(* IEC 61131-3 sources: SRCI/RobotLibrary/Library/POUs/General/MC_RobotTask (part 2) *)

END_METHOD

METHOD PRIVATE CreateSendPayload : DINT
VAR_IN_OUT
  /// Robot assignment of function
  AxesGroup                 : AxesGroup;
  /// Outputs of PLC for communication to RC
  RobotOutData              : ARRAY[0..RobotLibraryParameter.ROBOT_OUT_DATA_MAX] OF BYTE;
END_VAR

VAR
  /// internal index
 _idx                       : DINT;
  /// temporary byte
 _tmpByte                   : BYTE;
  /// internal sequence index
 _seqIdx                    : DINT;
  /// internal fragment index
 _fragIdx                   : DINT;
END_VAR

  // ------------------------------------
  // Fill SendData
  // ------------------------------------
  // reset all variables and payload
  SendData.Reset();

  CreateSendPayloadHeader        ( AxesGroup := AxesGroup );
  CreateSendPayloadCyclic        ( AxesGroup := AxesGroup );
  CreateSendPayloadCyclicOptional( AxesGroup := AxesGroup );
  CreateSendPayloadSequence      ( AxesGroup := AxesGroup );
  CreateSendPayloadFooter        ( AxesGroup := AxesGroup );
  CreateSendPayloadLogging       ( AxesGroup := AxesGroup );

  // Copy payload to outputs
  SysDepMemCpy( pDest := ADR(RobotOutData), pSrc := ADR(SendData.Payload), DataLen := RobotLibraryParameter.ROBOT_OUT_DATA_MAX+1);

  // reset NewSEQ flag
  AxesGroup.State.NewSEQ[0] := FALSE; {warning 'Test'}

END_METHOD

METHOD PRIVATE CreateSendPayloadCyclic : DINT
VAR_IN_OUT
  /// Robot assignment of function
  AxesGroup : AxesGroup;
END_VAR

  SendData.AddByte(Telegram.PlcToRob.Cyclic.ToolNo);
  SendData.AddByte(Telegram.PlcToRob.Cyclic.FrameNo);

END_METHOD

METHOD PRIVATE CreateSendPayloadCyclicOptional : DINT
VAR_IN_OUT
  /// Robot assignment of function
  AxesGroup : AxesGroup;
END_VAR

VAR
  /// temporary byte
 _tmpByte   : BYTE;
END_VAR

  // Telegram.PlcToRob.CyclicOptional.SubProgramData {{{
  IF ( AxesGroup.CyclicOptional.PlcToRob.SubProgramData.Active )
  THEN
    SendData.AddDataBlock( ADR(Telegram.PlcToRob.CyclicOptional.SubProgramData.Data), SIZEOF(Telegram.PlcToRob.CyclicOptional.SubProgramData.Data));
  END_IF
  // }}}

  // Telegram.PlcToRob.CyclicOptional.CartesianPos {{{
  IF ( AxesGroup.CyclicOptional.PlcToRob.CartesianPosition.Active)
  THEN
    SendData.AddReal(Telegram.PlcToRob.CyclicOptional.CartesianPosition.X );
    SendData.AddReal(Telegram.PlcToRob.CyclicOptional.CartesianPosition.Y );
    SendData.AddReal(Telegram.PlcToRob.CyclicOptional.CartesianPosition.Z );
    SendData.AddReal(Telegram.PlcToRob.CyclicOptional.CartesianPosition.Rx);
    SendData.AddReal(Telegram.PlcToRob.CyclicOptional.CartesianPosition.Ry);
    SendData.AddReal(Telegram.PlcToRob.CyclicOptional.CartesianPosition.Rz);

   _tmpByte   := 0;
   _tmpByte.0 := Telegram.PlcToRob.CyclicOptional.CartesianPosition.Config.0;
   _tmpByte.1 := Telegram.PlcToRob.CyclicOptional.CartesianPosition.Config.1;
   _tmpByte.2 := Telegram.PlcToRob.CyclicOptional.CartesianPosition.Config.2;

    SendData.AddByte(_tmpByte);

    SendData.AddByte (Telegram.PlcToRob.CyclicOptional.CartesianPosition.Turns_J2_J1             );
    SendData.AddByte (Telegram.PlcToRob.CyclicOptional.CartesianPosition.Turns_J4_J3             );
    SendData.AddByte (Telegram.PlcToRob.CyclicOptional.CartesianPosition.Turns_J6_J5             );
    SendData.AddByte (Telegram.PlcToRob.CyclicOptional.CartesianPosition.Turns_E1                );
    SendData.AddReal (Telegram.PlcToRob.CyclicOptional.CartesianPosition.E1                      );
  END_IF
  // }}}

  // Telegram.PlcToRob.CyclicOptional.JointPosition {{{
  IF ( AxesGroup.CyclicOptional.PlcToRob.JointPosition.Active)
  THEN
    SendData.AddReal(Telegram.PlcToRob.CyclicOptional.JointPosition.J1);
    SendData.AddReal(Telegram.PlcToRob.CyclicOptional.JointPosition.J2);
    SendData.AddReal(Telegram.PlcToRob.CyclicOptional.JointPosition.J3);
    SendData.AddReal(Telegram.PlcToRob.CyclicOptional.JointPosition.J4);
    SendData.AddReal(Telegram.PlcToRob.CyclicOptional.JointPosition.J5);
    SendData.AddReal(Telegram.PlcToRob.CyclicOptional.JointPosition.J6);
    SendData.AddReal(Telegram.PlcToRob.CyclicOptional.JointPosition.E1);
  END_IF
  // }}}

  // Telegram.PlcToRob.CyclicOptional.Force {{{
  IF ( AxesGroup.CyclicOptional.PlcToRob.Force.Active)
  THEN
    SendData.AddReal(Telegram.PlcToRob.CyclicOptional.Force.X);
    SendData.AddReal(Telegram.PlcToRob.CyclicOptional.Force.Y);
    SendData.AddReal(Telegram.PlcToRob.CyclicOptional.Force.Z);
    SendData.AddReal(Telegram.PlcToRob.CyclicOptional.Force.Rx);
    SendData.AddReal(Telegram.PlcToRob.CyclicOptional.Force.Ry);
    SendData.AddReal(Telegram.PlcToRob.CyclicOptional.Force.Rz);
  END_IF
  // }}}

  // Telegram.PlcToRob.CyclicOptional.TwoSequences {{{
  // }}}

  // AxesGroup.OptionalCyclic.PlcToRob.CartesianPosExt {{{
  IF ( AxesGroup.CyclicOptional.PlcToRob.CartesianPositionExt.Active)
  THEN
    SendData.AddReal(Telegram.PlcToRob.CyclicOptional.CartesianPositionExt.E2);
    SendData.AddReal(Telegram.PlcToRob.CyclicOptional.CartesianPositionExt.E3);
    SendData.AddReal(Telegram.PlcToRob.CyclicOptional.CartesianPositionExt.E4);
    SendData.AddReal(Telegram.PlcToRob.CyclicOptional.CartesianPositionExt.E5);
    SendData.AddReal(Telegram.PlcToRob.CyclicOptional.CartesianPositionExt.E6);
  END_IF
  // }}}

  // AxesGroup.OptionalCyclic.PlcToRob.JointPositionExt {{{
  IF ( AxesGroup.CyclicOptional.PlcToRob.JointPositionExt.Active)
  THEN
    SendData.AddReal(Telegram.PlcToRob.CyclicOptional.JointPositionExt.E2);
    SendData.AddReal(Telegram.PlcToRob.CyclicOptional.JointPositionExt.E3);
    SendData.AddReal(Telegram.PlcToRob.CyclicOptional.JointPositionExt.E4);
    SendData.AddReal(Telegram.PlcToRob.CyclicOptional.JointPositionExt.E5);
    SendData.AddReal(Telegram.PlcToRob.CyclicOptional.JointPositionExt.E6);
  END_IF
  // }}}

  // Telegram.PlcToRob.CyclicOptional..CartesianForceExt {{{
  IF ( AxesGroup.CyclicOptional.PlcToRob.ForceExt.Active)
  THEN
    SendData.AddReal(Telegram.PlcToRob.CyclicOptional.ForceExt.E1);
    SendData.AddReal(Telegram.PlcToRob.CyclicOptional.ForceExt.E2);
    SendData.AddReal(Telegram.PlcToRob.CyclicOptional.ForceExt.E3);
    SendData.AddReal(Telegram.PlcToRob.CyclicOptional.ForceExt.E4);
    SendData.AddReal(Telegram.PlcToRob.CyclicOptional.ForceExt.E5);
    SendData.AddReal(Telegram.PlcToRob.CyclicOptional.ForceExt.E6);
  END_IF
  // }}}

END_METHOD

METHOD PRIVATE CreateSendPayloadFooter : DINT
VAR_IN_OUT
  /// Robot assignment of function
  AxesGroup : AxesGroup;
END_VAR
VAR
  /// index of lifesign in footer
  _lifeSignIdxFooter : DINT;
END_VAR

  IF (( _parCfg.Com.TelegramLengthPlcToRob    >= 1                                           ) AND
      ( _parCfg.Com.TelegramLengthPlcToRob    <= RobotLibraryParameter.ROBOT_OUT_DATA_MAX +1 ))
  THEN
    // set index of life sign byte
   _lifeSignIdxFooter := _parCfg.Com.TelegramLengthPlcToRob -1;

    SendData.Payload[_lifeSignIdxFooter] := AxesGroup.Cyclic.PlcToRob.LifeSign;
  END_IF

END_METHOD

METHOD PRIVATE CreateSendPayloadHeader : DINT
VAR_IN_OUT
  /// Robot assignment of function
  AxesGroup : AxesGroup;
END_VAR

  SendData.AddByte(Telegram.PlcToRob.Header.SRCIVersion           );
  SendData.AddByte(Telegram.PlcToRob.Header.FastStop_LifeSign     );
  SendData.AddUint(Telegram.PlcToRob.Header.TelegramLengthPlcToRob);
  SendData.AddUint(Telegram.PlcToRob.Header.TelegramLengthRobToPlc);
  SendData.AddByte(Telegram.PlcToRob.Header.AxesGroupID_Control   );
  SendData.AddByte(Telegram.PlcToRob.Header.Reserved              );
  SendData.AddUint(Telegram.PlcToRob.Header.TelegramNumberPlcToRob);
  SendData.AddUint(Telegram.PlcToRob.Header.TelegramNumberRobToPlc);
  SendData.AddUint(Telegram.PlcToRob.Header.ClientDate            );
  SendData.AddTime(Telegram.PlcToRob.Header.ClientTime            );

END_METHOD

METHOD PRIVATE CreateSendPayloadLogging : DINT
VAR_IN_OUT
  /// Robot assignment of function
  AxesGroup                 : AxesGroup;
END_VAR

  IF  ((( Telegram.PlcToRob.Sequence[0].Header.PayloadLength > 0 ) AND (AxesGroup.State.NewSEQ[0] )) OR
       (( Telegram.PlcToRob.Sequence[1].Header.PayloadLength > 0 ) AND (AxesGroup.State.NewSEQ[1] )))
  THEN
    // Create log entry
    CreateLogMessagePara1 ( Timestamp   := SystemTime,
                            MessageType := MessageType.CMD,
                            Severity    := Severity.DEBUG,
                            MessageCode := 0,
                            MessageText := 'SendData: Bytes send in total: {1}',
                            Para1       :=  UDINT_TO_STRING(SendData.PayloadLen));
  END_IF

END_METHOD

METHOD PRIVATE CreateSendPayloadSequence : DINT
VAR_IN_OUT
  /// Robot assignment of function
  AxesGroup                 : AxesGroup;
END_VAR

VAR
  /// internal sequence index
 _seqIdx                    : DINT;
  /// internal fragment index
 _fragIdx                   : DINT;
END_VAR

  FOR _seqIdx := 0 TO AxesGroup.State.SequenceCountSend
  DO
    // Check 2nd sequence ? -> goto 2nd sequence payload address
    IF ( _seqIdx = SECONDARY_SEQUENCE )
    THEN
      SendData.PayloadPtr := CalculateSequencePayloadStartAdr(AxesGroup := AxesGroup,
                                                              Direction := ComDirection.PLC_TO_ROB,
                                                              Sequence  := SequenceFlag.SECONDARY_SEQUENCE);
    END_IF

    // Telegram.PlcToRob.Sequence[x].Header {{{
    SendData.AddUint(Telegram.PlcToRob.Sequence[_seqIdx].Header.SEQ_ACK);
    SendData.AddUint(Telegram.PlcToRob.Sequence[_seqIdx].Header.PayloadLength);
    // }}}

    // check limit reachted ?
    IF ( SendData.PayloadPtr + FOOTER_SIZE >= Telegram.PlcToRob.Header.TelegramLengthPlcToRob)
    THEN
      EXIT;
    END_IF

    // PlcToRob.Sequence[x].Fragment[x] {{{
    FOR _fragIdx := 0 TO AxesGroup.State.FragmentCountSend[_seqIdx]
    DO

      IF (Telegram.PlcToRob.Sequence[_seqIdx].Fragment[_fragIdx].Header.PayloadLength > 0)
      THEN
        // PlcToRob.Sequence[x].Fragment[x].Header {{{
        SendData.AddUint(Telegram.PlcToRob.Sequence[_seqIdx].Fragment[_fragIdx].Header.CmdID);
        SendData.AddByte(Telegram.PlcToRob.Sequence[_seqIdx].Fragment[_fragIdx].Header.Reserve);
        SendData.AddByte(Telegram.PlcToRob.Sequence[_seqIdx].Fragment[_fragIdx].Header.FragmentAction);
        SendData.AddUint(Telegram.PlcToRob.Sequence[_seqIdx].Fragment[_fragIdx].Header.PayloadPointer);
        SendData.AddUint(Telegram.PlcToRob.Sequence[_seqIdx].Fragment[_fragIdx].Header.PayloadLength);
        // }}}

        // PlcToRob.Sequence[x].Fragment[x].Command {{{

        // Hint: the command header is part of the fragment payload
        IF (Telegram.PlcToRob.Sequence[_seqIdx].Fragment[_fragIdx].Header.PayloadLength > 0)
        THEN
          SendData.AddDataBlock( pValue :=  ADR(Telegram.PlcToRob.Sequence[_seqIdx].Fragment[_fragIdx].Command.Payload           ) + Telegram.PlcToRob.Sequence[_seqIdx].Fragment[_fragIdx].Header.PayloadPointer,
                                   Size :=     (Telegram.PlcToRob.Sequence[_seqIdx].Fragment[_fragIdx].Header.PayloadLength      ));

        END_IF

        IF (SendData.PayloadLen = 232)
        THEN
          SendData.PayloadLen := SendData.PayloadLen;
  			END_IF

      END_IF
      // }}}
    END_FOR
    // }}}
  END_FOR

END_METHOD

METHOD FB_init : BOOL
VAR_INPUT
  bInitRetains : BOOL; // if TRUE, the retain variables are initialized (warm start / cold start)
  bInCopyCode : BOOL;  // if TRUE, the instance afterwards gets moved into the copy code (online change)
END_VAR

  MyType := 'MC_RobotTaskFB';

  // Create log entry
  CreateLogMessage ( Timestamp   := SystemTime,
                     MessageType := MessageType.CMD,
                     Severity    := Severity.DEBUG,
                     MessageCode := 0,
                     MessageText := 'PLC started / restarted');

END_METHOD

METHOD PRIVATE HandleAliveBit
VAR_INPUT
  LifeSign : BYTE;
END_VAR

VAR_INST
  /// flag that indicates that the 1st cyclce is running
  First : BOOL := TRUE;
END_VAR

  IF (First AND LifeSign > 0)
  THEN
    // init alive value
   _aliveValue := LifeSign;
    // reset first flag
    First := FALSE;
  END_IF

  _aliveCheck ( IN  := (_aliveValue = LifeSign) , PT := ParCfg.Com.LifeSignTimeOut + ParCfg.Plc.CycleTime);
  _alive_R    ( CLK := _aliveBit);
  _alive_F    ( CLK := _aliveBit);

  IF ( _aliveValue <> LifeSign)
  THEN
   _aliveValue := LifeSign;
   _aliveBit   := TRUE;
  END_IF

  IF (_aliveCheck.Q)
  THEN
   _aliveBit := FALSE;
  END_IF

  IF (_alive_R.Q)
  THEN
    // Create log entry
    CreateLogMessage ( Timestamp   := SystemTime,
                       MessageType := MessageType.CMD,
                       Severity    := Severity.INFO,
                       MessageCode := 0,
                       MessageText := 'Data Exchange is running (Alive-Bit)');
  END_IF

  IF (_alive_F.Q)
  THEN
    // Create log entry
    CreateLogMessage ( Timestamp   := SystemTime,
                       MessageType := MessageType.CMD,
                       Severity    := Severity.INFO,
                       MessageCode := 0,
                       MessageText := 'Data Exchange has stopped (Alive-Bit)');
  END_IF

END_METHOD

METHOD PRIVATE HandleAxesGroup
VAR_IN_OUT
  /// Robot assignment of function
  AxesGroup : AxesGroup;
END_VAR

  HandleAxesGroupAcyclic       ( AxesGroup    := AxesGroup);
  HandleAxesGroupCyclic        ( AxesGroup    := AxesGroup);
  HandleAxesGroupCyclicOptional( AxesGroup    := AxesGroup);
  HandleAxesGroupMessageLog    ( AxesGroup    := AxesGroup);
  HandleAxesGroupParameter     ( AxesGroup    := AxesGroup);
  HandleAxesGroupState         ( AxesGroup    := AxesGroup);

END_METHOD

METHOD PRIVATE HandleAxesGroupAcyclic
VAR_IN_OUT
  /// Robot assignment of function
  AxesGroup : AxesGroup;
END_VAR

  // Call active command register FB
  AxesGroup.Acyclic.ActiveCommandRegister(SystemTime     := SystemTime,
                                          RegisterSize   := MIN( RobotLibraryParameter.ACTIVE_CMD_REGISTER_ENTRIES_MAX, AxesGroup.Parameter.Rob.Parameter.LengthACR),
                                          InternalLogger := AxesGroup.MessageLog,
                                          ExternalLogger := AxesGroup.MessageLog.ExternalLogger,
                                          LogLevel       := AxesGroup.MessageLog.LogLevel);

END_METHOD

METHOD PRIVATE HandleAxesGroupCyclic
VAR_IN_OUT
  /// Robot assignment of function
  AxesGroup : AxesGroup;
END_VAR

  // set instance AxesGroupID
  AxesGroup.Cyclic.PlcToRob.AxesGroupID := AxesGroupID;
  // Set Version
  AxesGroup.Cyclic.PlcToRob.SRCIVersion := RobotLibraryConstants.SRCIVersion;

  AxesGroup.Cyclic.PlcToRob.TelegramLengthPlcToRob := _parCfg.Com.TelegramLengthPlcToRob;
  AxesGroup.Cyclic.PlcToRob.TelegramLengthRobToPlc := _parCfg.Com.TelegramLengthRobToPlc;

  AxesGroup.Cyclic.PlcToRob.TelegramNumberPlcToRob := PlcOptionalCyclicToUint(AxesGroup.Parameter.Plc.OptionalCyclic);
  AxesGroup.Cyclic.PlcToRob.TelegramNumberRobToPlc := RobOptionalCyclicToUint(AxesGroup.Parameter.Rob.OptionalCyclic);

  // Set Date + Time
  AxesGroup.Cyclic.PlcToRob.ClientDate  := DATE_TO_IEC_DATE(SystemTime.SystemDate);
  AxesGroup.Cyclic.PlcToRob.ClientTime  := TIME_TO_IEC_TIME(SystemTime.SystemTime);

END_METHOD

METHOD PRIVATE HandleAxesGroupCyclicOptional
VAR_IN_OUT
  /// Robot assignment of function
  AxesGroup : AxesGroup;
END_VAR

  // PlcToRob {{{
  AxesGroup.CyclicOptional.PlcToRob.SubProgramData      .Active := AxesGroup.Parameter.Plc.OptionalCyclic.UseCallSubprogram;
  AxesGroup.CyclicOptional.PlcToRob.CartesianPosition   .Active := AxesGroup.Parameter.Plc.OptionalCyclic.UseCartesianPosition;
  AxesGroup.CyclicOptional.PlcToRob.JointPosition       .Active := AxesGroup.Parameter.Plc.OptionalCyclic.UseJointPosition;
  AxesGroup.CyclicOptional.PlcToRob.Force               .Active := AxesGroup.Parameter.Plc.OptionalCyclic.UseForce;
  AxesGroup.CyclicOptional.PlcToRob.CartesianPositionExt.Active := AxesGroup.Parameter.Plc.OptionalCyclic.UseCartesianPositionExt;
  AxesGroup.CyclicOptional.PlcToRob.JointPositionExt    .Active := AxesGroup.Parameter.Plc.OptionalCyclic.UseJointPositionExt;
  // }}}

  // RobToPlc {{{
  AxesGroup.CyclicOptional.RobToPlc.SubProgramData      .Active := AxesGroup.Parameter.Rob.OptionalCyclic.UseCallSubprogram;
  AxesGroup.CyclicOptional.RobToPlc.CartesianPosition   .Active := AxesGroup.Parameter.Rob.OptionalCyclic.UseCartesianPosition;
  AxesGroup.CyclicOptional.RobToPlc.JointPosition       .Active := AxesGroup.Parameter.Rob.OptionalCyclic.UseJointPosition;
  AxesGroup.CyclicOptional.RobToPlc.Force               .Active := AxesGroup.Parameter.Rob.OptionalCyclic.UseForce;
  AxesGroup.CyclicOptional.RobToPlc.Current             .Active := AxesGroup.Parameter.Rob.OptionalCyclic.UseCurrent;
  AxesGroup.CyclicOptional.RobToPlc.CartesianPositionExt.Active := AxesGroup.Parameter.Rob.OptionalCyclic.UseCartesianPositionExt;
  AxesGroup.CyclicOptional.RobToPlc.JointPositionExt    .Active := AxesGroup.Parameter.Rob.OptionalCyclic.UseJointPositionExt;
  AxesGroup.CyclicOptional.RobToPlc.ForceExt            .Active := AxesGroup.Parameter.Rob.OptionalCyclic.UseForceExt;
  AxesGroup.CyclicOptional.RobToPlc.CurrentExt          .Active := AxesGroup.Parameter.Rob.OptionalCyclic.UseCurrentExt;
  // }}}

END_METHOD

METHOD PRIVATE HandleAxesGroupMessageLog
VAR_IN_OUT
  /// Robot assignment of function
  AxesGroup  : AxesGroup;
END_VAR

  // Set External logger
  AxesGroup.MessageLog.ExternalLogger := ExternalLogger;
  AxesGroup.MessageLog.LogLevel       := LogLevel;

  IF (AxesGroup.State.GroupReset_R.Q)
  THEN
    AxesGroup.MessageLog.DeleteMessages();
    AxesGroup.MessageLog.DeleteSystemLogs();
  END_IF

END_METHOD

METHOD PRIVATE HandleAxesGroupParameter
VAR_IN_OUT
  /// Robot assignment of function
  AxesGroup : AxesGroup;
END_VAR

  IF (_exchangeConfiguration.Enabled)
  THEN
    AxesGroup.Parameter.Plc.Parameter                           := _parCfg.Plc.Parameter;
    AxesGroup.Parameter.Plc.OptionalCyclic                      := _parCfg.Plc.OptionalCyclic;
    AxesGroup.Parameter.Rob.OptionalCyclic                      := _parCfg.Rob.OptionalCyclic;

    AxesGroup.Parameter.Rob.Parameter.LengthACR                 := _exchangeConfiguration.OutCmd.LengthACR;
    AxesGroup.Parameter.Rob.Parameter.HighestToolIndex          := _exchangeConfiguration.OutCmd.HighestToolIndex;
    AxesGroup.Parameter.Rob.Parameter.HighestFrameIndex         := _exchangeConfiguration.OutCmd.HighestFrameIndex;
    AxesGroup.Parameter.Rob.Parameter.HighestLoadIndex          := _exchangeConfiguration.OutCmd.HighestLoadIndex;
    AxesGroup.Parameter.Rob.Parameter.HighestWorkAreaIndex      := _exchangeConfiguration.OutCmd.HighestWorkAreaIndex;
    AxesGroup.Parameter.Rob.Parameter.DataInSync                := _exchangeConfiguration.OutCmd.DataInSync;
    AxesGroup.Parameter.Rob.Parameter.ChangeIndexTool           := _exchangeConfiguration.OutCmd.ChangeIndexTool;
    AxesGroup.Parameter.Rob.Parameter.ChangeIndexFrame          := _exchangeConfiguration.OutCmd.ChangeIndexFrame;
    AxesGroup.Parameter.Rob.Parameter.ChangeIndexLoad           := _exchangeConfiguration.OutCmd.ChangeIndexLoad;
    AxesGroup.Parameter.Rob.Parameter.ChangeIndexWorkArea       := _exchangeConfiguration.OutCmd.ChangeIndexWorkArea;
    AxesGroup.Parameter.Rob.Parameter.RAWorkingHours            := _exchangeConfiguration.OutCmd.RAWorkingHours;
    AxesGroup.Parameter.Rob.Parameter.BrakeTestRequired         := _exchangeConfiguration.OutCmd.BrakeTestRequired;
    AxesGroup.Parameter.Rob.Parameter.StepModeExactStopActive   := _exchangeConfiguration.OutCmd.StepModeExactStopActive;
    AxesGroup.Parameter.Rob.Parameter.StepModeBlendingActive    := _exchangeConfiguration.OutCmd.StepModeBlendingActive;
    AxesGroup.Parameter.Rob.Parameter.PathAccuracyMode          := _exchangeConfiguration.OutCmd.PathAccuracyMode;
    AxesGroup.Parameter.Rob.Parameter.AvoidSingularity          := _exchangeConfiguration.OutCmd.AvoidSingularity;
    AxesGroup.Parameter.Rob.Parameter.CollisionDetectionEnabled := _exchangeConfiguration.OutCmd.CollisionDetectionEnabled;
    AxesGroup.Parameter.Rob.Parameter.AcceleratingSupported     := _exchangeConfiguration.OutCmd.AcceleratingSupported;
    AxesGroup.Parameter.Rob.Parameter.DecceleratingSupported    := _exchangeConfiguration.OutCmd.DecceleratingSupported;
    AxesGroup.Parameter.Rob.Parameter.ConstantVelocitySupported := _exchangeConfiguration.OutCmd.ConstantVelocitySupported;
    AxesGroup.Parameter.Rob.Parameter.RCWorkingHours            := _exchangeConfiguration.OutCmd.RCWorkingHours;
  ELSE
    AxesGroup.Parameter.Plc.Parameter                           := ParCfg.Plc.Parameter;
    AxesGroup.Parameter.Plc.OptionalCyclic                      := ParCfg.Plc.OptionalCyclic;
    AxesGroup.Parameter.Rob.OptionalCyclic                      := ParCfg.Rob.OptionalCyclic;
  END_IF

END_METHOD

METHOD PRIVATE HandleAxesGroupState
VAR_IN_OUT
  /// Robot assignment of function
  AxesGroup : AxesGroup;
END_VAR
VAR
  /// internal index for loops
 _idx       : DINT;
END_VAR

  AxesGroup.State.AliveOk      := _aliveBit;
  AxesGroup.State.Initialized  := Initialized  AND AxesGroup.State.AliveOk;
  AxesGroup.State.Synchronized := Synchronized AND AxesGroup.State.AliveOk;
  AxesGroup.State.CMDsEnabled  := AxesGroup.State.Initialized OR
                                  AxesGroup.State.Synchronized;

  AxesGroup.State.ConfigExchanged := _exchangeConfiguration.Enabled;

  AxesGroup.State.UnifiedFrameIndex                    := DINT_TO_USINT( MIN( RobotLibraryParameter.FRAME_MAX -1    , _exchangeConfiguration.OutCmd.HighestFrameIndex   ));
  AxesGroup.State.UnifiedToolIndex                     := DINT_TO_USINT( MIN( RobotLibraryParameter.TOOL_MAX -1     , _exchangeConfiguration.OutCmd.HighestToolIndex    ));
  AxesGroup.State.UnifiedLoadIndex                     := DINT_TO_USINT( MIN( RobotLibraryParameter.LOAD_MAX-1      , _exchangeConfiguration.OutCmd.HighestLoadIndex    ));
  AxesGroup.State.UnifiedWorkAreaIndex                 := DINT_TO_USINT( MIN( RobotLibraryParameter.WORK_AREAS_MAX-1, _exchangeConfiguration.OutCmd.HighestWorkAreaIndex));

  AxesGroup.State.DataEnableSync                       := _exchangeConfiguration.ParCmd.DataEnableSync;
  AxesGroup.State.SyncStateRc.InSync.Frame             := _exchangeConfiguration.OutCmd.DataInSync.FramesInSync;
  AxesGroup.State.SyncStateRc.InSync.Tool              := _exchangeConfiguration.OutCmd.DataInSync.ToolsInSync;
  AxesGroup.State.SyncStateRc.InSync.Load              := _exchangeConfiguration.OutCmd.DataInSync.LoadsInSync;
  AxesGroup.State.SyncStateRc.InSync.WorkArea          := _exchangeConfiguration.OutCmd.DataInSync.WorkAreasInSync;
  AxesGroup.State.SyncStateRc.InSync.SwLimits          := _exchangeConfiguration.OutCmd.DataInSync.SoftwareLimitsInSync;
  AxesGroup.State.SyncStateRc.InSync.DefaultDynamics   := _exchangeConfiguration.OutCmd.DataInSync.DefaultDynamicsInSync;
  AxesGroup.State.SyncStateRc.InSync.ReferenceDynamics := _exchangeConfiguration.OutCmd.DataInSync.ReferenceDynamicsInSync;

  AxesGroup.State.SyncStateRc.UnSyncNo.Frame           := _exchangeConfiguration.OutCmd.ChangeIndexFrame;
  AxesGroup.State.SyncStateRc.UnSyncNo.Tool            := _exchangeConfiguration.OutCmd.ChangeIndexTool;
  AxesGroup.State.SyncStateRc.UnSyncNo.Load            := _exchangeConfiguration.OutCmd.ChangeIndexLoad;
  AxesGroup.State.SyncStateRc.UnSyncNo.WorkArea        := _exchangeConfiguration.OutCmd.ChangeIndexWorkArea;

  // Update internal data
  AxesGroup.State.SystemTime   := SystemTime;
  AxesGroup.State.OnlineChange := OnlineChange;
  AxesGroup.State.Initialized  := Initialized;

  // Create rising and falling edges for Online Change
  AxesGroup.State.OnlineChange_R(CLK := OnlineChange);
  AxesGroup.State.OnlineChange_F(CLK := OnlineChange);

  // Create rising and falling edges for GroupReset
  AxesGroup.State.GroupReset_R(CLK := AxesGroup.State.GroupReset);
  AxesGroup.State.GroupReset_F(CLK := AxesGroup.State.GroupReset);

  // Copy function block results
  AxesGroup.State.RobotData         := _readRobotData.OutCmd;
  AxesGroup.State.ConfigurationData := _exchangeConfiguration.OutCmd;

END_METHOD

METHOD PRIVATE HandleInvalidFrames
VAR_IN_OUT
   /// Robot assignment of function
  AxesGroup   : AxesGroup;
    /// Inputs of PLC for communication from RC
  RobotInData : ARRAY[0..RobotLibraryParameter.ROBOT_IN_DATA_MAX ] OF BYTE;
END_VAR
VAR
  /// index of lifesign in header
 _lifeSignIdxHeader : DINT;
  /// Value of lifesign in header
 _lifeSignHeader    : BYTE;
  /// index of lifesign in footer
 _lifeSignIdxFooter : DINT;
  /// Value of lifesign in footer
 _lifeSignFooter    : BYTE;
END_VAR
VAR_INST
  /// Timeout for invalid frames counter check
 _invalidFrameCounterCheck_D : TON;
  /// last count of invalid frames
 _lastInvalidFrames          : UDINT;
END_VAR

  IF (( _parCfg.Com.TelegramLengthRobToPlc     < 1                                       ) AND
      ( _parCfg.Com.TelegramLengthRobToPlc - 1 > RobotLibraryParameter.ROBOT_IN_DATA_MAX ))
  THEN
    // no valid telegram length settings
    RETURN;
  END_IF

  // set index of last byte
  _lifeSignIdxHeader := 1;
  _lifeSignIdxFooter := _parCfg.Com.TelegramLengthRobToPlc -1;

  IF ( AxesGroup.Cyclic.RobToPlc.TelegramState = TelegramState.INITIALIZED )
  THEN
    // Get lifesign values
   _lifeSignHeader := GetHalfeByteHi( RobotInData[_lifeSignIdxHeader]);
   _lifeSignFooter := GetHalfeByteHi( RobotInData[_lifeSignIdxFooter]);
  END_IF

  // Timer for invalid frame(s) message
  _invalidFrameCounterCheck_D( IN := TRUE , PT := RobotLibraryParameter.INVALID_FRAMES_CHECK_TIMEOUT);

  // Check Frame is valid :
  // ----------------------
  IF ( _lifeSignHeader <> _lifeSignFooter )
  THEN
    AxesGroup.State.InvalidFrames := AxesGroup.State.InvalidFrames + 1;
  END_IF

  // Check timeout for invalid frame message
  IF ( _invalidFrameCounterCheck_D.Q )
  THEN
    // reset timer
   _invalidFrameCounterCheck_D( IN := FALSE);

    // compare invalid frame(s) counter
    IF ( AxesGroup.State.InvalidFrames <> _lastInvalidFrames)
    THEN
      // store last invalid frame(s) counter value
     _lastInvalidFrames := AxesGroup.State.InvalidFrames;
      // Create log entry
      CreateLogMessagePara1 ( Timestamp   := SystemTime,
                              MessageType := MessageType.CMD,
                              Severity    := Severity.WARNING,
                              MessageCode := 0,
                              MessageText := 'Detected invalid frames {1} in total',
                              Para1       :=  UDINT_TO_STRING(AxesGroup.State.InvalidFrames));
    END_IF
  END_IF

  // Reset invalid frames counter with rising edge of group reset
  IF ( AxesGroup.State.GroupReset_R.Q)
  THEN
    AxesGroup.State.InvalidFrames := 0;
               _lastInvalidFrames := 0;

    // Create log entry
    CreateLogMessage ( Timestamp   := SystemTime,
                       MessageType := MessageType.CMD,
                       Severity    := Severity.INFO,
                       MessageCode := 0,
                       MessageText := 'Reset invalid frames counter by executing GroupReset');
  END_IF

END_METHOD

METHOD PRIVATE HandleLifeSign
VAR_IN_OUT
  /// Robot assignment of function
  AxesGroup    : AxesGroup;
END_VAR
VAR_INST
  /// flag for 1st cycle
 _first : BOOL := TRUE;
END_VAR

  IF ( _first ) OR ( NOT Enable )
  THEN
    // init LifeSign
    AxesGroup.Cyclic.PlcToRob.LifeSign := 0;
    // reset first flag
   _first := FALSE;
    // prevent inc LifeSign in the 1st cycle (Code below)
    RETURN;
  END_IF

  AxesGroup.Cyclic.PlcToRob.LifeSign := AxesGroup.Cyclic.PlcToRob.LifeSign + 1;

  IF ( AxesGroup.Cyclic.PlcToRob.LifeSign > 15 )
  THEN
    AxesGroup.Cyclic.PlcToRob.LifeSign := 1; // 0 is only in the very 1st cycle to indicate the system start in logging
  END_IF

  IF ( Enable ) AND ( _alive_F.Q )
  THEN
    // Reset initialized flag
    Initialized := FALSE;
    // Reset Synchronized flag
    Synchronized := FALSE;

    // Set error
    ErrorID := RobotLibraryErrorIdEnum.ERR_CONNECTION_LOST;
    // Create log entry
    CreateLogMessage ( Timestamp   := SystemTime,
                       MessageType := MessageType.CMD,
                       Severity    := Severity.FATAL_ERROR,
                       MessageCode := 0,
                       MessageText := 'LifeSign timeout -> Reinitialization required !');
  END_IF

  // Reset connection lost error
  IF ( NOT Enable ) AND ( _aliveBit ) AND ( ErrorID = RobotLibraryErrorIdEnum.ERR_CONNECTION_LOST )
  THEN
    ErrorID := 0;
  END_IF

END_METHOD

METHOD HandleLogMessagesAck
VAR_IN_OUT
   /// Robot assignment of function
  AxesGroup : AxesGroup;
END_VAR

  IF (( _readMessages.Enabled           ) AND
      ( _readMessages.OutCmd.MsgId > 0  ))
  THEN
    // Check if message has been entered into the message log ?
    IF ( AxesGroup.MessageLog.CheckMessageCodePresent(_readMessages.OutCmd.ErrorCode ))
    THEN
      // Set Message ID as Acknowlege ID
     _readMessages.ParCmd.MsgID := _readMessages.OutCmd.MsgId;
  	END_IF
  END_IF

END_METHOD

METHOD PRIVATE HandleSeqAck
VAR_IN_OUT
   /// Robot assignment of function
  AxesGroup    : AxesGroup;
END_VAR
VAR
  /// internal index for loops
 _idx : DINT;
END_VAR

  FOR _idx := 0 TO  AxesGroup.State.SequenceCountSend
  DO
    AxesGroup.State.CurrentAck[_idx] := Telegram.RobToPlc.Sequence[_idx].Header.SEQ_ACK;

    IF (NOT Enable)
    THEN
      AxesGroup.State.CurrentSEQ[0] := 0;
      AxesGroup.State.CurrentSEQ[1] := 0;
    END_IF

    // Check Seq/Ack :
    // ----------------------
    IF ( AxesGroup.State.CurrentAck[_idx] = AxesGroup.State.CurrentSEQ[_idx] )
    THEN
      AxesGroup.State.CurrentSEQ[_idx] := MAX(AxesGroup.State.CurrentSEQ[0],AxesGroup.State.CurrentSEQ[1]) +1;

      IF (AxesGroup.State.CurrentSEQ[_idx] >= 255) {warning 'ToDo: Test for Yaskawa'}
      THEN
        AxesGroup.State.CurrentSEQ[_idx] := 0;
  		END_IF

      AxesGroup.State.NewSEQ[_idx] := TRUE;
    END_IF
  END_FOR

END_METHOD

METHOD PRIVATE HandleSync
VAR_IN_OUT
   /// Robot assignment of function
  AxesGroup : AxesGroup;
  /// ToolData stored on PLC.For more information refer to 5.5.6.4
  ToolData          : ARRAY[0..RobotLibraryParameter.TOOL_MAX -1      ] OF Tool;
  /// LoadData stored on PLC.For more information refer to 5.5.6.4
  FrameData         : ARRAY[0..RobotLibraryParameter.FRAME_MAX -1     ] OF Frame;
  /// LoadData stored on PLC.For more information refer to 5.5.6.4
  LoadData          : ARRAY[0..RobotLibraryParameter.LOAD_MAX -1      ] OF Load;
  /// Work areas stored on PLC. For more information refer to 5.5.8
  WorkAreas         : ARRAY[0..RobotLibraryParameter.WORK_AREAS_MAX -1] OF RobotWorkArea;
  /// Software limits stored on PLC
  SWLimits          : SWLimits;
  /// Default dynamics stored on PLC. For more information refer to 5.5.7
  DefaultDynamics   : DefaultDynamics;
  /// Reference dynamics stored on PLC. For more information refer to 5.5.7
  ReferenceDynamics : ReferenceDynamics;
END_VAR

VAR
  /// flag that indicates at least any iten has enabled synchronisation
 _dataEnableSyncAny        : BOOL;
  /// flag that indicates that the frame datas are synchronized or deactivated
 _inSyncFrameOk            : BOOL;
  /// flag that indicates that the tool datas are synchronized or deactivated
 _inSyncToolOk             : BOOL;
  /// flag that indicates that the load datas are synchronized or deactivated
 _inSyncLoadOk             : BOOL;
  /// flag that indicates that the work areas are synchronized or deactivated
 _inSyncWorkAreaOk         : BOOL;
  /// flag that indicates that the SW limits are synchronized or deactivated
 _inSyncSwLimitsOk         : BOOL;
  /// flag that indicates that the default dynamice are synchronized or deactivated
 _inSyncDefaultDynamicOk   : BOOL;
  /// flag that indicates that the reference dynamice are synchronized or deactivated
 _InSyncReferenceDynamicOk : BOOL;
END_VAR

  HandleSyncToolData              ( AxesGroup := AxesGroup, ToolData          := ToolData);
  //RETURN; {warning 'ToDo: Enable Sync again'}

  HandleSyncFrameData             ( AxesGroup := AxesGroup, FrameData         := FrameData);
  HandleSyncLoadData              ( AxesGroup := AxesGroup, LoadData          := LoadData);
  HandleSyncRobotDefaultDynamics  ( AxesGroup := AxesGroup, DefaultDynamics   := DefaultDynamics);
  HandleSyncRobotReferenceDynamics( AxesGroup := AxesGroup, ReferenceDynamics := ReferenceDynamics);
  HandleSyncRobotSWLimits         ( AxesGroup := AxesGroup, SwLimits          := SwLimits);
  HandleSyncToolData              ( AxesGroup := AxesGroup, ToolData          := ToolData);
  HandleSyncWorkArea              ( AxesGroup := AxesGroup, WorkAreas         := WorkAreas);

  // check any synchronisation activated ?
  _dataEnableSyncAny :=        ((     AxesGroup.State.DataEnableSync.EnableSyncFrame             )  OR
                                (     AxesGroup.State.DataEnableSync.EnableSyncTool              )  OR
                                (     AxesGroup.State.DataEnableSync.EnableSyncLoad              )  OR
                                (     AxesGroup.State.DataEnableSync.EnableSyncWorkArea          )  OR
                                (     AxesGroup.State.DataEnableSync.EnableSyncSWLimits          )  OR
                                (     AxesGroup.State.DataEnableSync.EnableSyncDefaultDynamics   )  OR
                                (     AxesGroup.State.DataEnableSync.EnableSyncReferenceDynamics ));

  _inSyncFrameOk :=            ((     AxesGroup.State.SyncStatePlc     .InSync.Frame             )  AND
                                (     AxesGroup.State.SyncStateRc      .InSync.Frame             )) OR
                                ( NOT AxesGroup.State.DataEnableSync.EnableSyncFrame             );

  _inSyncToolOk :=             ((     AxesGroup.State.SyncStatePlc     .InSync.Tool              )  AND
                                (     AxesGroup.State.SyncStateRc      .InSync.Tool              )) OR
                                ( NOT AxesGroup.State.DataEnableSync.EnableSyncTool              );

  _inSyncLoadOk :=             ((     AxesGroup.State.SyncStatePlc     .InSync.Load              )  AND
                                (     AxesGroup.State.SyncStateRc      .InSync.Load              )) OR
                                ( NOT AxesGroup.State.DataEnableSync.EnableSyncLoad              );

  _inSyncWorkAreaOk :=         ((     AxesGroup.State.SyncStatePlc     .InSync.WorkArea          )  AND
                                (     AxesGroup.State.SyncStateRc      .InSync.WorkArea          )) OR
                                ( NOT AxesGroup.State.DataEnableSync.EnableSyncWorkArea          );

  _inSyncSwLimitsOk :=         ((     AxesGroup.State.SyncStatePlc    .InSync.SwLimits           )  AND
                                (     AxesGroup.State.SyncStateRc      .InSync.SwLimits          )) OR
                                ( NOT AxesGroup.State.DataEnableSync.EnableSyncSwLimits          );

  _inSyncDefaultDynamicOk :=   ((     AxesGroup.State.SyncStatePlc     .InSync.DefaultDynamics   )  AND
                                (     AxesGroup.State.SyncStateRc      .InSync.DefaultDynamics   )) OR
                                ( NOT AxesGroup.State.DataEnableSync.EnableSyncDefaultDynamics   );

  _inSyncReferenceDynamicOk := ((     AxesGroup.State.SyncStatePlc     .InSync.ReferenceDynamics )  AND
                                (     AxesGroup.State.SyncStateRc      .InSync.ReferenceDynamics )) OR
                                ( NOT AxesGroup.State.DataEnableSync.EnableSyncReferenceDynamics );

  Synchronized := (( _inSyncFrameOk            ) AND
                   ( _inSyncToolOk             ) AND
                   ( _inSyncLoadOk             ) AND
                   ( _inSyncWorkAreaOk         ) AND
                   ( _inSyncSwLimitsOk         ) AND
                   ( _inSyncDefaultDynamicOk   ) AND
                   ( _InSyncReferenceDynamicOk ) AND
                   ( _dataEnableSyncAny        ));

  // Update exchange configuration parameter
  _exchangeConfiguration.ParCmd.DataInSync.FramesInSync            := AxesGroup.State.SyncStatePlc.InSync.Frame;
  _exchangeConfiguration.ParCmd.DataInSync.ToolsInSync             := AxesGroup.State.SyncStatePlc.InSync.Tool;
  _exchangeConfiguration.ParCmd.DataInSync.LoadsInSync             := AxesGroup.State.SyncStatePlc.InSync.Load;
  _exchangeConfiguration.ParCmd.DataInSync.WorkAreasInSync         := AxesGroup.State.SyncStatePlc.InSync.WorkArea;
  _exchangeConfiguration.ParCmd.DataInSync.SoftwareLimitsInSync    := AxesGroup.State.SyncStatePlc.InSync.SwLimits;
  _exchangeConfiguration.ParCmd.DataInSync.DefaultDynamicsInSync   := AxesGroup.State.SyncStatePlc.InSync.DefaultDynamics;
  _exchangeConfiguration.ParCmd.DataInSync.ReferenceDynamicsInSync := AxesGroup.State.SyncStatePlc.InSync.ReferenceDynamics;

END_METHOD

METHOD PRIVATE HandleSyncFrameData
VAR_IN_OUT
   /// Robot assignment of function
  AxesGroup : AxesGroup;
  /// FrameData stored on PLC.For more information refer to 5.5.6.4
  FrameData : ARRAY[0..RobotLibraryParameter.FRAME_MAX -1] OF Frame;
END_VAR

VAR
  /// Internal step counter name
 _stepName        : STRING;
  /// Internal reference to step counter
 _rStep           : REFERENCE TO DINT;
  /// Internal reference to timer
 _rTimer          : REFERENCE TO TON;
  /// Internal reference to timeout
 _rTimeout        : REFERENCE TO TIME;
  /// Internal reference to synchroniztion index
 _rSyncIdx        : REFERENCE TO USINT;
  /// internal bit for condition found
 _found           : BOOL;
  /// empty data set to reset all DataChanged bits
 _dataChangedNone : AxesGroupStateDataChanged;
END_VAR

  // Set internal references
  _stepName      :=   '_stepSyncFrameData = ';
  _rStep       REF=    _stepSyncFrameData;
  _rTimer      REF=   _timerSyncFrameData;
  _rTimeout    REF= _timeoutSyncFrameData;
  _rSyncIdx    REF=     _syncIdxFrameData;

  CASE _rStep
  OF
    0: // Check initialisation configured ?
       IF (( _parCfg.PLC.Parameter.SynchronizationModes.Frame[SyncTime.DURING_START_UP] = SyncMode.NO_SYNCHRONIZATION ) AND
           ( _parCfg.PLC.Parameter.SynchronizationModes.Frame[SyncTime. AFTER_START_UP] = SyncMode.NO_SYNCHRONIZATION ))
       THEN
         RETURN;
       END_IF

       // wait for initialisation done
       IF  ((     AxesGroup.State.RobotData.RCSupportedFunctions. ReadFrameData ) AND
            (     AxesGroup.State.RobotData.RCSupportedFunctions.WriteFrameData ) AND
            (     AxesGroup.State.Initialized                                   ) AND
            ( NOT Error                                                         ))
       THEN
         // Check PLC frames < RC frames and SyncFrame enabled ?
         IF (( AxesGroup.State.DataEnableSync.EnableSyncFrame      = TRUE                              )  AND
             ( AxesGroup.Parameter.Rob.Parameter.HighestFrameIndex > RobotLibraryParameter.FRAME_MAX -1 ))
         THEN
           WarningID := RobotLibraryWarningIdEnum.WARN_FRAME_DATA_ARRAY_TOO_SHORT;
         END_IF

         // Create log entry
         CreateLogMessagePara1 ( Timestamp   := SystemTime,
                                 MessageType := MessageType.CMD,
                                 Severity    := Severity.DEBUG,
                                 MessageCode := 0,
                                 MessageText := 'SyncFrameData: Start initial reading of FrameData from RC',
                                 Para1       :=  '');

         // init frame number
        _rSyncIdx := 0;
         // init count of unsynchronized elements
         AxesGroup.State.SyncStatePlc.UnSyncNo.Frame := 0;
         // set timeout
         SetTimeout(PT := _rTimeout, rTimer := _rTimer);
         // inc step counter
        _rStep := _rStep + 1;
       END_IF

       // Start read FrameData
    1: IF (( NOT _readFrameData.Busy  ) AND
           ( NOT _readFrameData.Error ))
       THEN
         // set command parameter
        _readFrameData.ParCmd.FrameNo := _rSyncIdx;
         // execute command
        _readFrameData.Execute := TRUE;
         // set timeout
         SetTimeout(PT := _rTimeout, rTimer := _rTimer);
         // inc step counter
        _rStep := _rStep + 1;
       ELSE
         // check error ?
         IF ( _readFrameData.Error ) AND ( WarningID = RobotLibraryWarningIdEnum.NO_WARNING )
         THEN
           WarningID := RobotLibraryWarningIdEnum.WARN_FRAME_SYNC_FAILED_BY_ERROR_OF_READ_OR_WRITE_CMD;
         END_IF

         // timeout exceeded ?
         IF (CheckTimeout(_rTimer) = RobotLibraryConstants.OK)
         THEN
           ErrorID     := RobotLibraryErrorIdEnum.ERR_TIMEOUT_CMD;
           ErrorAddTxt := CONCAT(_stepName, DINT_TO_STRING(_rStep));
         END_IF
       END_IF

       // Wait Framedata read
    2: IF (( NOT _readFrameData.Busy  ) AND
           ( NOT _readFrameData.Error ) AND
           (     _readFrameData.Done  ))
       THEN
         // reset execution
        _readFrameData.Execute := FALSE;
         // set available bit
        _frameData[_rSyncIdx].Available := TRUE;
         FrameData[_rSyncIdx].Available := TRUE;
         // Copy data
        _frameData[_rSyncIdx].Data := _readFrameData.OutCmd.FrameData;

         // Check frame data is equal ?
         IF ( NOT IsFrameDataEqual( Data1 := _frameData[_rSyncIdx].Data, Data2 := FrameData[_rSyncIdx].Data, IgnoreTimestamp := TRUE))
         THEN
           // Reset plc in sync flag
           AxesGroup.State.SyncStatePlc.InSync.Frame := FALSE;
           // Set data changed flag
           AxesGroup.State.DataChanged.Frame[_rSyncIdx] := TRUE;
           // inc count of unsynchronised plc frames
           AxesGroup.State.SyncStatePlc.UnSyncNo.Frame := AxesGroup.State.SyncStatePlc.UnSyncNo.Frame + 1;

           // Create log entry
           CreateLogMessagePara1 ( Timestamp   := SystemTime,
                                   MessageType := MessageType.CMD,
                                   Severity    := Severity.DEBUG,
                                   MessageCode := 0,
                                   MessageText := 'SyncFrameData: Detected a difference in Frame[{1}] between PLC and RC',
                                   Para1       :=  DINT_TO_STRING(_rSyncIdx));

           // Check synchronisation is enabled ?
           IF ( NOT AxesGroup.State.DataEnableSync.EnableSyncFrame ) AND (InfoID = RobotLibraryInfoIdEnum.NO_INFO )
           THEN
             InfoID := RobotLibraryInfoIdEnum.INFO_SYNC_FRAME_DATA_DISABLED;
  				 END_IF

           // Check user interaction needed ?
           IF ( AxesGroup.Parameter.PLC.Parameter.SyncUserInteraction.Frame ) AND ( WarningID = RobotLibraryWarningIdEnum.NO_WARNING )
           THEN
             WarningID := RobotLibraryWarningIdEnum.WARN_FRAME_NUMBER_SYNC_ERROR;
  				 END_IF
  			 END_IF

         // Check all frames read ?
         IF ( _rSyncIdx < AxesGroup.State.UnifiedFrameIndex )
         THEN
           // set timeout
           SetTimeout(PT := _rTimeout, rTimer := _rTimer);
           // inc frame index
          _rSyncIdx := _rSyncIdx + 1;
           // dec step counter
          _rStep := _rStep - 1;
         ELSE
           // set timeout
           SetTimeout(PT := _rTimeout, rTimer := _rTimer);
           // inc step counter
          _rStep := _rStep + 1;
         END_IF
       ELSE
         // check error ?
         IF (_readFrameData.Error)
         THEN
           // Set warning
           WarningID := RobotLibraryWarningIdEnum.WARN_FRAME_SYNC_FAILED_BY_ERROR_OF_READ_OR_WRITE_CMD;
           // reset available bit
           FrameData[_rSyncIdx].Available := FALSE;
          _frameData[_rSyncIdx].Available := FALSE;
         END_IF

         // timeout exceeded ?
         IF (CheckTimeout(_rTimer) = RobotLibraryConstants.OK)
         THEN
           ErrorID     := RobotLibraryErrorIdEnum.ERR_TIMEOUT_CMD;
           ErrorAddTxt := CONCAT(_stepName, DINT_TO_STRING(_rStep));
         END_IF
       END_IF

       // Check synchronisation state ?
    3: IF (( AxesGroup.State.SyncStatePlc.UnSyncNo.Frame                                            = 0                           ) OR
           ( AxesGroup.Parameter.Plc.Parameter.SynchronizationModes.Frame[SyncTime.DURING_START_UP] = SyncMode.NO_SYNCHRONIZATION ))
       THEN
         // Update bit for data in sync
         AxesGroup.State.SyncStatePlc.InSync.Frame := (AxesGroup.State.SyncStatePlc.UnSyncNo.Frame = 0);
         // set timeout
         SetTimeout(PT := _rTimeout, rTimer := _rTimer);
         // inc step counter
        _rStep := 10; // -> jump to after startup

         // Create log entry
         CreateLogMessagePara1 ( Timestamp   := SystemTime,
                                 MessageType := MessageType.CMD,
                                 Severity    := Severity.DEBUG,
                                 MessageCode := 0,
                                 MessageText := 'SyncFrameData: Synchronization Startup Phase done',
                                 Para1       :=  '' );
       ELSE
         // Check user interaction needed ?
         IF ( NOT AxesGroup.Parameter.PLC.Parameter.SyncUserInteraction.Frame )
         THEN
           CASE AxesGroup.Parameter.Plc.Parameter.SynchronizationModes.Frame[SyncTime.DURING_START_UP] OF

             SyncMode.SERVER_TO_CLIENT :

               // Overwrite PLC data with RC data
               FrameData := _frameData;
               // Reset data changed flags
               AxesGroup.State.DataChanged.Frame := _dataChangedNone.Frame;
               // Reset Synchronizing flag
               AxesGroup.State.Synchronizing.Frame := FALSE;
               // Set plc in sync flag
               AxesGroup.State.SyncStatePlc.InSync.Frame := TRUE;
               // Reset count of unsynchronised plc frames
               AxesGroup.State.SyncStatePlc.UnSyncNo.Frame := 0;
               // set timeout
               SetTimeout(PT := _rTimeout, rTimer := _rTimer);
               // inc step counter
              _rStep := 10; // -> jump to after startup

              // Create log entry
              CreateLogMessagePara3 ( Timestamp   := SystemTime,
                                      MessageType := MessageType.CMD,
                                      Severity    := Severity.DEBUG,
                                      MessageCode := 0,
                                      MessageText := 'SyncFrameData: Synchronization of Frames triggered by StartUp-Compare, SyncMode = {2}, SyncTime = {3}, SyncDirection = RC -> PLC',
                                      Para1       :=  DINT_TO_STRING(_rSyncIdx),
                                      Para2       :=  SYNC_MODE_TO_STRING(AxesGroup.Parameter.Plc.Parameter.SynchronizationModes.Frame[SyncTime.DURING_START_UP]),
                                      Para3       :=  SYNC_TIME_TO_STRING(SyncTime.DURING_START_UP));
              // Create log entry
              CreateLogMessagePara1 ( Timestamp   := SystemTime,
                                      MessageType := MessageType.CMD,
                                      Severity    := Severity.DEBUG,
                                      MessageCode := 0,
                                      MessageText := 'SyncFrameData: Applied the initial read frame data from RC',
                                      Para1       :=  '' );

  				   SyncMode.CLIENT_TO_SERVER : ;

               // Check conflicts to solve ?
               FOR _rSyncIdx := 0 TO AxesGroup.State.UnifiedFrameIndex
               DO
                 IF ( AxesGroup.State.DataChanged.Frame[_rSyncIdx] )
                 THEN
                  _found := TRUE;
                   EXIT;
  		  			   END_IF
               END_FOR

               IF ( _found )
               THEN
                 // Reset plc in sync flag
                 AxesGroup.State.SyncStatePlc.InSync.Frame := FALSE;
                 // Set Synchronizing flag
                 AxesGroup.State.Synchronizing.Frame := TRUE;
                 // set timeout
                 SetTimeout(PT := _rTimeout, rTimer := _rTimer);
                 // inc step counter
                _rStep := _rStep +1; // -> write PLC data to RC
                 // Create log entry
                 CreateLogMessagePara3 ( Timestamp   := SystemTime,
                                         MessageType := MessageType.CMD,
                                         Severity    := Severity.DEBUG,
                                         MessageCode := 0,
                                         MessageText := 'SyncFrameData: Synchronization of Frame[{1}] triggered by StartUp-Compare, SyncMode = {2}, SyncTime = {3}, SyncDirection = PLC -> RC',
                                         Para1       :=  DINT_TO_STRING(_rSyncIdx),
                                         Para2       :=  SYNC_MODE_TO_STRING(AxesGroup.Parameter.Plc.Parameter.SynchronizationModes.Frame[SyncTime.DURING_START_UP]),
                                         Para3       :=  SYNC_TIME_TO_STRING(SyncTime.DURING_START_UP));
               ELSE
                 // Reset data changed flags
                 AxesGroup.State.DataChanged.Frame := _dataChangedNone.Frame;
                 // Reset Synchronizing flag
                 AxesGroup.State.Synchronizing.Frame := FALSE;
                 // Set plc in sync flag
                 AxesGroup.State.SyncStatePlc.InSync.Frame := TRUE;
                 // Reset count of unsynchronised frames
                 AxesGroup.State.SyncStatePlc.UnSyncNo.Frame := 0;
                 // set timeout
                 SetTimeout(PT := _rTimeout, rTimer := _rTimer);
                 // inc step counter
                _rStep := 10; // -> jump to after startup
  				     END_IF
           ELSE
             // invalid sync mode for startup
             ErrorID := RobotLibraryErrorIdEnum.ERR_SYNC_MODE_INVALID;
   	       END_CASE
         END_IF
       END_IF

       // Start write frame data
    4: IF (( NOT _writeFrameData.Busy  ) AND
           ( NOT _writeFrameData.Error ))
       THEN
         // set command parameter
        _writeFrameData.ParCmd.FrameNo   := _rSyncIdx;
        _writeFrameData.ParCmd.FrameData :=  FrameData[_rSyncIdx].Data;
         // execute command
        _writeFrameData.Execute := TRUE;
         // set timeout
         SetTimeout(PT := _rTimeout, rTimer := _rTimer);
         // inc step counter
        _rStep := _rStep + 1;
       ELSE
         // check error ?
         IF (_writeFrameData.Error)
         THEN
           ErrorID     := _writeFrameData.ErrorID;
           ErrorAddTxt := _writeFrameData.ErrorAddTxt;;
         END_IF

         // timeout exceeded ?
         IF (CheckTimeout(_rTimer) = RobotLibraryConstants.OK)
         THEN
           ErrorID     := RobotLibraryErrorIdEnum.ERR_TIMEOUT_CMD;
           ErrorAddTxt := CONCAT(_stepName, DINT_TO_STRING(_rStep));
         END_IF
       END_IF

       // Wait frame data written ?
    5: IF (( NOT _writeFrameData.Busy  ) AND
           ( NOT _writeFrameData.Error ) AND
           (     _writeFrameData.Done  ))
       THEN
         // execute command
        _writeFrameData.Execute := FALSE;
         // apply frame data to internal frame data
        _frameData[_rSyncIdx] := FrameData[_rSyncIdx];
         // reset data changed bit
         AxesGroup.State.DataChanged.Frame[_rSyncIdx] := FALSE;
         // dec count of unsynchronised frames
         AxesGroup.State.SyncStatePlc.UnSyncNo.Frame := AxesGroup.State.SyncStatePlc.UnSyncNo.Frame - 1;
         // set timeout
         SetTimeout(PT := _rTimeout, rTimer := _rTimer);
         // dec step counter
        _rStep := _rStep - 2;
       ELSE
         // check error ?
         IF (_writeFrameData.Error)
         THEN
           WarningID := RobotLibraryWarningIdEnum.WARN_FRAME_SYNC_FAILED_BY_ERROR_OF_READ_OR_WRITE_CMD;
         END_IF

         // timeout exceeded ?
         IF (CheckTimeout(_rTimer) = RobotLibraryConstants.OK)
         THEN
           ErrorID     := RobotLibraryErrorIdEnum.ERR_TIMEOUT_CMD;
           ErrorAddTxt := CONCAT(_stepName, DINT_TO_STRING(_rStep));
         END_IF
       END_IF

    // --------------------------------------------
    // SyncMode after startup :
    // --------------------------------------------

    10 : // check synchronisation active ?
         IF ( AxesGroup.Parameter.Plc.Parameter.SynchronizationModes.Frame[SyncTime.AFTER_START_UP] = SyncMode.NO_SYNCHRONIZATION)
         THEN
           RETURN;
         END_IF

         // reset count of unsynchronised frames
         AxesGroup.State.SyncStatePlc.UnSyncNo.Frame := 0;

         // Check all frame datas
         FOR _rSyncIdx := 0 TO AxesGroup.State.UnifiedFrameIndex
         DO
           // compare frame data
           AxesGroup.State.DataChanged.Frame[_rSyncIdx] := NOT IsFrameDataEqual( Data1 := FrameData[_rSyncIdx].Data, Data2 := _frameData[_rSyncIdx].Data, IgnoreTimestamp := FALSE);

           // Check Frame data changed ?
           IF (AxesGroup.State.DataChanged.Frame[_rSyncIdx])
           THEN
             // inc count of unsynchronised plc frames
             AxesGroup.State.SyncStatePlc.UnSyncNo.Frame := AxesGroup.State.SyncStatePlc.UnSyncNo.Frame + 1;
             // Create log entry
             CreateLogMessagePara2 ( Timestamp   := SystemTime,
                                     MessageType := MessageType.CMD,
                                     Severity    := Severity.DEBUG,
                                     MessageCode := 0,
                                     MessageText := 'SyncFrameData: Detected a local change of Frame[{1}] on PLC, SyncTime = {2}',
                                     Para1       :=  DINT_TO_STRING(_rSyncIdx),
                                     Para2       :=  SYNC_TIME_TO_STRING(SyncTime.AFTER_START_UP));
  				 END_IF

           // Update plc in sync flag
           AxesGroup.State.SyncStatePlc.InSync.Frame := (AxesGroup.State.SyncStatePlc.UnSyncNo.Frame = 0);
  	     END_FOR

         // Check synchronization is needed ?
         IF ( NOT AxesGroup.State.SyncStatePlc.InSync.Frame ) XOR
            ( NOT AxesGroup.State.SyncStateRc .InSync.Frame )
         THEN
           CASE AxesGroup.Parameter.Plc.Parameter.SynchronizationModes.Frame[SyncTime.AFTER_START_UP]
           OF
             // NO_SYNCHRONIZATION
             SyncMode.NO_SYNCHRONIZATION : ; // no further action

             // CLIENT_TO_SERVER
             SyncMode.CLIENT_TO_SERVER :
               // set timeout
               SetTimeout(PT := _rTimeout, rTimer := _rTimer);
               // inc step counter
              _rStep := 11;

             // SERVER_TO_CLIENT
             SyncMode.SERVER_TO_CLIENT :
               // set timeout
               SetTimeout(PT := _rTimeout, rTimer := _rTimer);
               // inc step counter
              _rStep := 12;

             // AUTOMATIC
             SyncMode.AUTOMATIC :
               // set timeout
               SetTimeout(PT := _rTimeout, rTimer := _rTimer);
               // inc step counter
              _rStep := 13;
           END_CASE
         ELSE
           // datas changeḍ on both sides ? -> Warning
           IF (( NOT AxesGroup.State.SyncStatePlc.InSync.Frame ) AND
               ( NOT AxesGroup.State.SyncStateRc .InSync.Frame ))
           THEN
             WarningID := RobotLibraryWarningIdEnum.WARN_FRAME_SYNC_BOTH_SIDES_CHANGED;
           END_IF
         END_IF

    // ------------------------------------------
    // SyncMode : CLIENT_TO_SERVER
    // ------------------------------------------
    11 : // Conflict triggerd by PLC ?
         IF ( NOT AxesGroup.State.SyncStatePlc.InSync.Frame )
         THEN
           // search for changed index
           FOR _rSyncIdx := 0 TO AxesGroup.State.UnifiedFrameIndex
           DO
             IF ( AxesGroup.State.DataChanged.Frame[_rSyncIdx] )
             THEN
               // set timeout
               SetTimeout(PT := _rTimeout, rTimer := _rTimer);
               // inc step counter
              _rStep := 30; // -> write PLC data to RC
               EXIT;
  					 END_IF
           END_FOR

           // Create log entry
           CreateLogMessagePara3 ( Timestamp   := SystemTime,
                                   MessageType := MessageType.CMD,
                                   Severity    := Severity.DEBUG,
                                   MessageCode := 0,
                                   MessageText := 'SyncFrameData: Synchronization of Frame[{1}] triggered by PLC, SyncMode = {2}, SyncTime = {3}, SyncDirection = PLC -> RC',
                                   Para1       :=  DINT_TO_STRING(_rSyncIdx),
                                   Para2       :=  SYNC_MODE_TO_STRING(AxesGroup.Parameter.Plc.Parameter.SynchronizationModes.Frame[SyncTime.AFTER_START_UP]),
                                   Para3       :=  SYNC_TIME_TO_STRING(SyncTime.AFTER_START_UP));
                                   RETURN;
         END_IF

         // Conflict triggered by RC ?
         IF ( NOT AxesGroup.State.SyncStateRc.InSync.Frame )
         THEN
           // get changed index
          _rSyncIdx := LIMIT(0, AxesGroup.State.SyncStateRc.UnSyncNo.Frame, AxesGroup.State.UnifiedFrameIndex);
           // set timeout
           SetTimeout(PT := _rTimeout, rTimer := _rTimer);
           // inc step counter
          _rStep := 30; // -> write PLC data to RC

           // Create log entry
           CreateLogMessagePara3 ( Timestamp   := SystemTime,
                                   MessageType := MessageType.CMD,
                                   Severity    := Severity.DEBUG,
                                   MessageCode := 0,
                                   MessageText := 'SyncFrameData: Synchronization of Frame[{1}] triggered by RC, SyncMode = {2}, SyncTime = {3}, SyncDirection = PLC -> RC',
                                   Para1       :=  DINT_TO_STRING(_rSyncIdx),
                                   Para2       :=  SYNC_MODE_TO_STRING(AxesGroup.Parameter.Plc.Parameter.SynchronizationModes.Frame[SyncTime.AFTER_START_UP]),
                                   Para3       :=  SYNC_TIME_TO_STRING(SyncTime.AFTER_START_UP));
                                   RETURN;
  			 END_IF

         // set timeout
         SetTimeout(PT := _rTimeout, rTimer := _rTimer);
         // jump back
        _rStep := 10;

    // ------------------------------------------
    // SyncMode : SERVER_TO_CLIENT
    // ------------------------------------------
    12 : // Conflict triggerd by PLC ?
         IF ( NOT AxesGroup.State.SyncStatePlc.InSync.Frame )
         THEN
           // search for changed index
           FOR _rSyncIdx := 0 TO AxesGroup.State.UnifiedFrameIndex
           DO
             IF ( AxesGroup.State.DataChanged.Frame[_rSyncIdx] )
             THEN
               // set timeout
               SetTimeout(PT := _rTimeout, rTimer := _rTimer);
               // inc step counter
              _rStep := 20; // -> read RC data and write it to PLC
               EXIT;
  					 END_IF
           END_FOR

           // Create log entry
           CreateLogMessagePara3 ( Timestamp   := SystemTime,
                                   MessageType := MessageType.CMD,
                                   Severity    := Severity.DEBUG,
                                   MessageCode := 0,
                                   MessageText := 'SyncFrameData: Synchronization of Frame[{1}] triggered by PLC, SyncMode = {2}, SyncTime = {3}, SyncDirection = RC -> PLC',
                                   Para1       :=  DINT_TO_STRING(_rSyncIdx),
                                   Para2       :=  SYNC_MODE_TO_STRING(AxesGroup.Parameter.Plc.Parameter.SynchronizationModes.Frame[SyncTime.AFTER_START_UP]),
                                   Para3       :=  SYNC_TIME_TO_STRING(SyncTime.AFTER_START_UP));
                                   RETURN;
         END_IF

         // Conflict triggered by RC ?
         IF ( NOT AxesGroup.State.SyncStateRc.InSync.Frame )
         THEN
           // get changed index
          _rSyncIdx := LIMIT(0, AxesGroup.State.SyncStateRc.UnSyncNo.Frame, AxesGroup.State.UnifiedFrameIndex);
           // set timeout
           SetTimeout(PT := _rTimeout, rTimer := _rTimer);
           // inc step counter
          _rStep := 20; // -> read RC data and write it to PLC

           // Create log entry
           CreateLogMessagePara3 ( Timestamp   := SystemTime,
                                   MessageType := MessageType.CMD,
                                   Severity    := Severity.DEBUG,
                                   MessageCode := 0,
                                   MessageText := 'SyncFrameData: Synchronization of Frame[{1}] triggered by RC, SyncMode = {2}, SyncTime = {3}, SyncDirection = RC -> PLC',
                                   Para1       :=  DINT_TO_STRING(_rSyncIdx),
                                   Para2       :=  SYNC_MODE_TO_STRING(AxesGroup.Parameter.Plc.Parameter.SynchronizationModes.Frame[SyncTime.AFTER_START_UP]),
                                   Para3       :=  SYNC_TIME_TO_STRING(SyncTime.AFTER_START_UP));
                                   RETURN;
  			 END_IF

         // set timeout
         SetTimeout(PT := _rTimeout, rTimer := _rTimer);
         // jump back
        _rStep := 10;

    // ------------------------------------------
    // SyncMode : AUTOMATIC
    // ------------------------------------------
    13 : // Conflict triggerd by PLC ?
         IF ( NOT AxesGroup.State.SyncStatePlc.InSync.Frame )
         THEN
           // search for changed index
           FOR _rSyncIdx := 0 TO AxesGroup.State.UnifiedFrameIndex
           DO
             IF ( AxesGroup.State.DataChanged.Frame[_rSyncIdx] )
             THEN
               // set timeout
               SetTimeout(PT := _rTimeout, rTimer := _rTimer);
               // inc step counter
              _rStep := 30; // -> write PLC data to RC
               EXIT;
  					 END_IF
           END_FOR

           // Create log entry
           CreateLogMessagePara3 ( Timestamp   := SystemTime,
                                   MessageType := MessageType.CMD,
                                   Severity    := Severity.DEBUG,
                                   MessageCode := 0,
                                   MessageText := 'SyncFrameData: Synchronization of Frame[{1}] triggered by PLC, SyncMode = {2}, SyncTime = {3}, SyncDirection = PLC -> RC',
                                   Para1       :=  DINT_TO_STRING(_rSyncIdx),
                                   Para2       :=  SYNC_MODE_TO_STRING(AxesGroup.Parameter.Plc.Parameter.SynchronizationModes.Frame[SyncTime.AFTER_START_UP]),
                                   Para3       :=  SYNC_TIME_TO_STRING(SyncTime.AFTER_START_UP));
                                   RETURN;
         END_IF

         // Conflict triggered by RC ?
         IF ( NOT AxesGroup.State.SyncStateRc.InSync.Frame )
         THEN
           // get changed index
          _rSyncIdx := LIMIT(0, AxesGroup.State.SyncStateRc.UnSyncNo.Frame, AxesGroup.State.UnifiedFrameIndex);
           // set timeout
           SetTimeout(PT := _rTimeout, rTimer := _rTimer);
           // inc step counter
          _rStep := 20; // -> read RC data an write it to PLC

           // Create log entry
           CreateLogMessagePara3 ( Timestamp   := SystemTime,
                                   MessageType := MessageType.CMD,
                                   Severity    := Severity.DEBUG,
                                   MessageCode := 0,
                                   MessageText := 'SyncFrameData: Synchronization of Frame[{1}] triggered by RC, SyncMode = {2}, SyncTime = {3}, SyncDirection = RC -> PLC',
                                   Para1       :=  DINT_TO_STRING(_rSyncIdx),
                                   Para2       :=  SYNC_MODE_TO_STRING(AxesGroup.Parameter.Plc.Parameter.SynchronizationModes.Frame[SyncTime.AFTER_START_UP]),
                                   Para3       :=  SYNC_TIME_TO_STRING(SyncTime.AFTER_START_UP));
                                   RETURN;
  			 END_IF

         // set timeout
         SetTimeout(PT := _rTimeout, rTimer := _rTimer);
         // jump back
        //_rStep := 10;

    // ------------------------------------------
    // Read Data from RC and write it to PLC
    // ------------------------------------------
    20 : IF (( NOT _readFrameData.Busy  ) AND
             ( NOT _readFrameData.Error ))
         THEN
           // set command parameter
          _readFrameData.ParCmd.FrameNo := _rSyncIdx;
           // execute command
          _readFrameData.Execute := TRUE;
           // set timeout
           SetTimeout(PT := _rTimeout, rTimer := _rTimer);
           // inc step counter
          _rStep := _rStep + 1;
         ELSE
           // check error ?
           IF (_readFrameData.Error)
           THEN
             ErrorID     := _readFrameData.ErrorID;
             ErrorAddTxt := _readFrameData.ErrorAddTxt;
           END_IF

           // timeout exceeded ?
           IF (CheckTimeout(_rTimer) = RobotLibraryConstants.OK)
           THEN
             ErrorID     := RobotLibraryErrorIdEnum.ERR_TIMEOUT_CMD;
             ErrorAddTxt := CONCAT(_stepName, DINT_TO_STRING(_rStep));
           END_IF
         END_IF

    21 : IF (( NOT _readFrameData.Busy  ) AND
             ( NOT _readFrameData.Error ) AND
             (     _readFrameData.Done  ))
         THEN
           // reset execution
          _readFrameData.Execute := FALSE;
           // update internal frame data
           FrameData[_rSyncIdx].Data := _readFrameData.OutCmd.FrameData;
          _frameData[_rSyncIdx].Data := _readFrameData.OutCmd.FrameData;
           // set available bit
           FrameData[_rSyncIdx].Available := TRUE;
          _frameData[_rSyncIdx].Available := TRUE;
           // set timeout
           SetTimeout(PT := _rTimeout, rTimer := _rTimer);
           // inc step counter
          _rStep := 10; // -> jump to after startup
         ELSE
           // check error ?
           IF (_readFrameData.Error)
           THEN
             ErrorID     := _readFrameData.ErrorID;
             ErrorAddTxt := _readFrameData.ErrorAddTxt;
             // reset available bit
             FrameData[_rSyncIdx].Available := FALSE;
            _frameData[_rSyncIdx].Available := FALSE;
           END_IF

           // timeout exceeded ?
           IF (CheckTimeout(_rTimer) = RobotLibraryConstants.OK)
           THEN
             ErrorID     := RobotLibraryErrorIdEnum.ERR_TIMEOUT_CMD;
             ErrorAddTxt := CONCAT(_stepName, DINT_TO_STRING(_rStep));
           END_IF
         END_IF

    // ------------------------------------------
    // Write data from PLC to RC
    // ------------------------------------------
    30 : IF (( NOT _writeFrameData.Busy  ) AND
             ( NOT _writeFrameData.Error ))
         THEN
           // set command parameter
          _writeFrameData.ParCmd.FrameNo   := _rSyncIdx;
          _writeFrameData.ParCmd.FrameData :=  FrameData[_rSyncIdx].Data;
           // execute command
          _writeFrameData.Execute := TRUE;
           // set timeout
           SetTimeout(PT := _rTimeout, rTimer := _rTimer);
           // inc step counter
          _rStep := _rStep + 1;
         ELSE
           // check error ?
           IF (_writeFrameData.Error)
           THEN
             ErrorID     := _writeFrameData.ErrorID;
             ErrorAddTxt := _writeFrameData.ErrorAddTxt;;
           END_IF

           // timeout exceeded ?
           IF (CheckTimeout(_rTimer) = RobotLibraryConstants.OK)
           THEN
             ErrorID     := RobotLibraryErrorIdEnum.ERR_TIMEOUT_CMD;
             ErrorAddTxt := CONCAT(_stepName, DINT_TO_STRING(_rStep));
           END_IF
         END_IF

    31 : IF (( NOT _writeFrameData.Busy  ) AND
             ( NOT _writeFrameData.Error ) AND
             (     _writeFrameData.Done  ))
         THEN
           // execute command
          _writeFrameData.Execute := FALSE;
           // update internal frame data
          _frameData[_rSyncIdx] := FrameData[_rSyncIdx];
           // set available bit
           FrameData[_rSyncIdx].Available := TRUE;
          _frameData[_rSyncIdx].Available := TRUE;
           // set timeout
           SetTimeout(PT := _rTimeout, rTimer := _rTimer);
           // inc step counter
          _rStep := 10; // -> jump to after startup;
         ELSE
           // check error ?
           IF (_writeFrameData.Error)
           THEN
             WarningID := RobotLibraryWarningIdEnum.WARN_FRAME_SYNC_FAILED_BY_ERROR_OF_READ_OR_WRITE_CMD;
             // reset available bit
             FrameData[_rSyncIdx].Available := FALSE;
            _frameData[_rSyncIdx].Available := FALSE;
           END_IF

           // timeout exceeded ?
           IF (CheckTimeout(_rTimer) = RobotLibraryConstants.OK)
           THEN
             ErrorID     := RobotLibraryErrorIdEnum.ERR_TIMEOUT_CMD;
             ErrorAddTxt := CONCAT(_stepName, DINT_TO_STRING(_rStep));
           END_IF
         END_IF

  ELSE
    // invalid step
    ErrorID     := RobotLibraryErrorIdEnum.ERR_INVALID_STEP;
    ErrorAddTxt := CONCAT(_stepName , DINT_TO_STRING(_stepCmd));
  END_CASE

END_METHOD

METHOD PRIVATE HandleSyncLoadData
VAR_IN_OUT
   /// Robot assignment of function
  AxesGroup : AxesGroup;
  /// LoadData stored on PLC.For more information refer to 5.5.6.4
  LoadData  : ARRAY[0..RobotLibraryParameter.LOAD_MAX -1] OF Load;
END_VAR

VAR
  /// Internal step counter name
 _stepName        : STRING;
  /// Internal reference to step counter
 _rStep           : REFERENCE TO DINT;
  /// Internal reference to timer
 _rTimer          : REFERENCE TO TON;
  /// Internal reference to timeout
 _rTimeout        : REFERENCE TO TIME;
  /// Internal reference to synchroniztion index
 _rSyncIdx        : REFERENCE TO USINT;
  /// internal bit for condition found
 _found           : BOOL;
  /// empty data set to reset all DataChanged bits
 _dataChangedNone : AxesGroupStateDataChanged;
END_VAR

  // Set internal references
  _stepName      :=   '_stepSyncLoadData = ';
  _rStep       REF=    _stepSyncLoadData;
  _rTimer      REF=   _timerSyncLoadData;
  _rTimeout    REF= _timeoutSyncLoadData;
  _rSyncIdx    REF=     _syncIdxLoadData;

  CASE _rStep
  OF
    0: // Check initialisation configured ?
       IF (( _parCfg.PLC.Parameter.SynchronizationModes.Load[SyncTime.DURING_START_UP] = SyncMode.NO_SYNCHRONIZATION ) AND
           ( _parCfg.PLC.Parameter.SynchronizationModes.Load[SyncTime. AFTER_START_UP] = SyncMode.NO_SYNCHRONIZATION ))
       THEN
         RETURN;
       END_IF

       // wait for initialisation done
       IF  ((     AxesGroup.State.RobotData.RCSupportedFunctions. ReadLoadData ) AND
            (     AxesGroup.State.RobotData.RCSupportedFunctions.WriteLoadData ) AND
            (     AxesGroup.State.Initialized                                  ) AND
            ( NOT Error                                                        ))
       THEN
         // Check PLC loads < RC Loads and SyncLoad enabled ?
         IF (( AxesGroup.State.DataEnableSync.EnableSyncLoad      = TRUE                              )  AND
             ( AxesGroup.Parameter.Rob.Parameter.HighestLoadIndex > RobotLibraryParameter.Load_MAX -1 ))
         THEN
           WarningID := RobotLibraryWarningIdEnum.WARN_LOAD_DATA_ARRAY_TOO_SHORT;
         END_IF

         // Create log entry
         CreateLogMessagePara1 ( Timestamp   := SystemTime,
                                 MessageType := MessageType.CMD,
                                 Severity    := Severity.DEBUG,
                                 MessageCode := 0,
                                 MessageText := 'SyncLoadData: Start initial reading of LoadData from RC',
                                 Para1       :=  '');

         // init load number
        _rSyncIdx := 1; //  !!! Attention : 0 is not allowed - LoadData starts with 1 !!!
         // init count of unsynchronized elements
         AxesGroup.State.SyncStatePlc.UnSyncNo.Load := 0;
         // set timeout
         SetTimeout(PT := _rTimeout, rTimer := _rTimer);
         // inc step counter
        _rStep := _rStep + 1;
       END_IF

       // Start read LoadData
    1: IF (( NOT _readLoadData.Busy  ) AND
           ( NOT _readLoadData.Error ))
       THEN
         // set command parameter
        _readLoadData.ParCmd.LoadNo := _rSyncIdx;
         // execute command
        _readLoadData.Execute := TRUE;
         // set timeout
         SetTimeout(PT := _rTimeout, rTimer := _rTimer);
         // inc step counter
        _rStep := _rStep + 1;
       ELSE
         // check error ?
         IF ( _readLoadData.Error ) AND ( WarningID = RobotLibraryWarningIdEnum.NO_WARNING )
         THEN
           WarningID := RobotLibraryWarningIdEnum.WARN_LOAD_SYNC_FAILED_BY_ERROR_OF_READ_OR_WRITE_CMD;
         END_IF

         // timeout exceeded ?
         IF (CheckTimeout(_rTimer) = RobotLibraryConstants.OK)
         THEN
           ErrorID     := RobotLibraryErrorIdEnum.ERR_TIMEOUT_CMD;
           ErrorAddTxt := CONCAT(_stepName, DINT_TO_STRING(_rStep));
         END_IF
       END_IF

       // Wait Loaddata read
    2: IF (( NOT _readLoadData.Busy  ) AND
           ( NOT _readLoadData.Error ) AND
           (     _readLoadData.Done  ))
       THEN
         // reset execution
        _readLoadData.Execute := FALSE;
         // set available bit
        _loadData[_rSyncIdx].Available := TRUE;
         LoadData[_rSyncIdx].Available := TRUE;
         // Copy data
        _loadData[_rSyncIdx].Data := _readLoadData.OutCmd.LoadData;

         // Check Load data is equal ?
         IF ( NOT IsLoadDataEqual( Data1 := _loadData[_rSyncIdx].Data, Data2 := LoadData[_rSyncIdx].Data, IgnoreTimestamp := TRUE))
         THEN
           // Reset plc in sync flag
           AxesGroup.State.SyncStatePlc.InSync.Load := FALSE;
           // Set data changed flag
           AxesGroup.State.DataChanged.Load[_rSyncIdx] := TRUE;
           // inc count of unsynchronised plc Loads
           AxesGroup.State.SyncStatePlc.UnSyncNo.Load := AxesGroup.State.SyncStatePlc.UnSyncNo.Load + 1;

           // Create log entry
           CreateLogMessagePara1 ( Timestamp   := SystemTime,
                                   MessageType := MessageType.CMD,
                                   Severity    := Severity.DEBUG,
                                   MessageCode := 0,
                                   MessageText := 'SyncLoadData: Detected a difference in Load[{1}] between PLC and RC',
                                   Para1       :=  DINT_TO_STRING(_rSyncIdx));

           // Check synchronisation is enabled ?
           IF ( NOT AxesGroup.State.DataEnableSync.EnableSyncLoad ) AND (InfoID = RobotLibraryInfoIdEnum.NO_INFO )
           THEN
             InfoID := RobotLibraryInfoIdEnum.INFO_SYNC_LOAD_DATA_DISABLED;
  				 END_IF

           // Check user interaction needed ?
           IF ( AxesGroup.Parameter.PLC.Parameter.SyncUserInteraction.Load ) AND ( WarningID = RobotLibraryWarningIdEnum.NO_WARNING )
           THEN
             WarningID := RobotLibraryWarningIdEnum.WARN_LOAD_NUMBER_SYNC_ERROR;
  				 END_IF
  			 END_IF

         // Check all Loads read ?
         IF ( _rSyncIdx < AxesGroup.State.UnifiedLoadIndex )
         THEN
           // set timeout
           SetTimeout(PT := _rTimeout, rTimer := _rTimer);
           // inc Load index
          _rSyncIdx := _rSyncIdx + 1;
           // dec step counter
          _rStep := _rStep - 1;
         ELSE
           // set timeout
           SetTimeout(PT := _rTimeout, rTimer := _rTimer);
           // inc step counter
          _rStep := _rStep + 1;
         END_IF
       ELSE
         // check error ?
         IF (_readLoadData.Error)
         THEN
           // Set warning
           WarningID := RobotLibraryWarningIdEnum.WARN_LOAD_SYNC_FAILED_BY_ERROR_OF_READ_OR_WRITE_CMD;
           // reset available bit
           LoadData[_rSyncIdx].Available := FALSE;
          _loadData[_rSyncIdx].Available := FALSE;
         END_IF

         // timeout exceeded ?
         IF (CheckTimeout(_rTimer) = RobotLibraryConstants.OK)
         THEN
           ErrorID     := RobotLibraryErrorIdEnum.ERR_TIMEOUT_CMD;
           ErrorAddTxt := CONCAT(_stepName, DINT_TO_STRING(_rStep));
         END_IF
       END_IF

       // Check synchronisation state ?
    3: IF (( AxesGroup.State.SyncStatePlc.UnSyncNo.Load                                            = 0                           ) OR
           ( AxesGroup.Parameter.Plc.Parameter.SynchronizationModes.Load[SyncTime.DURING_START_UP] = SyncMode.NO_SYNCHRONIZATION ))
       THEN
         // Update bit for data in sync
         AxesGroup.State.SyncStatePlc.InSync.Load := (AxesGroup.State.SyncStatePlc.UnSyncNo.Load = 0);
         // set timeout
         SetTimeout(PT := _rTimeout, rTimer := _rTimer);
         // inc step counter
        _rStep := 10; // -> jump to after startup

         // Create log entry
         CreateLogMessagePara1 ( Timestamp   := SystemTime,
                                 MessageType := MessageType.CMD,
                                 Severity    := Severity.DEBUG,
                                 MessageCode := 0,
                                 MessageText := 'SyncLoadData: Synchronization Startup Phase done',
                                 Para1       :=  '' );
       ELSE
         // Check user interaction needed ?
         IF ( NOT AxesGroup.Parameter.PLC.Parameter.SyncUserInteraction.Load )
         THEN
           CASE AxesGroup.Parameter.Plc.Parameter.SynchronizationModes.Load[SyncTime.DURING_START_UP] OF

             SyncMode.SERVER_TO_CLIENT :

               // Overwrite PLC data with RC data
               LoadData := _loadData;
               // Reset data changed flags
               AxesGroup.State.DataChanged.Load := _dataChangedNone.Load;
               // Reset Synchronizing flag
               AxesGroup.State.Synchronizing.Load := FALSE;
               // Set plc in sync flag
               AxesGroup.State.SyncStatePlc.InSync.Load := TRUE;
               // Reset count of unsynchronised plc Loads
               AxesGroup.State.SyncStatePlc.UnSyncNo.Load := 0;
               // set timeout
               SetTimeout(PT := _rTimeout, rTimer := _rTimer);
               // inc step counter
              _rStep := 10; // -> jump to after startup

              // Create log entry
              CreateLogMessagePara3 ( Timestamp   := SystemTime,
                                      MessageType := MessageType.CMD,
                                      Severity    := Severity.DEBUG,
                                      MessageCode := 0,
                                      MessageText := 'SyncLoadData: Synchronization of Loads triggered by StartUp-Compare, SyncMode = {2}, SyncTime = {3}, SyncDirection = RC -> PLC',
                                      Para1       :=  DINT_TO_STRING(_rSyncIdx),
                                      Para2       :=  SYNC_MODE_TO_STRING(AxesGroup.Parameter.Plc.Parameter.SynchronizationModes.Load[SyncTime.DURING_START_UP]),
                                      Para3       :=  SYNC_TIME_TO_STRING(SyncTime.DURING_START_UP));
              // Create log entry
              CreateLogMessagePara1 ( Timestamp   := SystemTime,
                                      MessageType := MessageType.CMD,
                                      Severity    := Severity.DEBUG,
                                      MessageCode := 0,
                                      MessageText := 'SyncLoadData: Applied the initial read Load data from RC',
                                      Para1       :=  '' );

  				   SyncMode.CLIENT_TO_SERVER : ;

               // Check conflicts to solve ?
               FOR _rSyncIdx := 1 TO AxesGroup.State.UnifiedLoadIndex //  !!! Attention : 0 is not allowed - LoadData starts with 1 !!!
               DO
                 IF ( AxesGroup.State.DataChanged.Load[_rSyncIdx] )
                 THEN
                  _found := TRUE;
                   EXIT;
  		  			   END_IF
               END_FOR

               IF ( _found )
               THEN
                 // Reset plc in sync flag
                 AxesGroup.State.SyncStatePlc.InSync.Load := FALSE;
                 // Set Synchronizing flag
                 AxesGroup.State.Synchronizing.Load := TRUE;
                 // set timeout
                 SetTimeout(PT := _rTimeout, rTimer := _rTimer);
                 // inc step counter
                _rStep := _rStep +1; // -> write PLC data to RC
                 // Create log entry
                 CreateLogMessagePara3 ( Timestamp   := SystemTime,
                                         MessageType := MessageType.CMD,
                                         Severity    := Severity.DEBUG,
                                         MessageCode := 0,
                                         MessageText := 'SyncLoadData: Synchronization of Load[{1}] triggered by StartUp-Compare, SyncMode = {2}, SyncTime = {3}, SyncDirection = PLC -> RC',
                                         Para1       :=  DINT_TO_STRING(_rSyncIdx),
                                         Para2       :=  SYNC_MODE_TO_STRING(AxesGroup.Parameter.Plc.Parameter.SynchronizationModes.Load[SyncTime.DURING_START_UP]),
                                         Para3       :=  SYNC_TIME_TO_STRING(SyncTime.DURING_START_UP));
               ELSE
                 // Reset data changed flags
                 AxesGroup.State.DataChanged.Load := _dataChangedNone.Load;
                 // Reset Synchronizing flag
                 AxesGroup.State.Synchronizing.Load := FALSE;
                 // Set plc in sync flag
                 AxesGroup.State.SyncStatePlc.InSync.Load := TRUE;
                 // Reset count of unsynchronised Loads
                 AxesGroup.State.SyncStatePlc.UnSyncNo.Load := 0;
                 // set timeout
                 SetTimeout(PT := _rTimeout, rTimer := _rTimer);
                 // inc step counter
                _rStep := 10; // -> jump to after startup
  				     END_IF
           ELSE
             // invalid sync mode for startup
             ErrorID := RobotLibraryErrorIdEnum.ERR_SYNC_MODE_INVALID;
   	       END_CASE
         END_IF
       END_IF

       // Start write Load data
    4: IF (( NOT _writeLoadData.Busy  ) AND
           ( NOT _writeLoadData.Error ))
       THEN
         // set command parameter
        _writeLoadData.ParCmd.LoadNo   := _rSyncIdx;
        _writeLoadData.ParCmd.LoadData :=  LoadData[_rSyncIdx].Data;
         // execute command
        _writeLoadData.Execute := TRUE;
         // set timeout
         SetTimeout(PT := _rTimeout, rTimer := _rTimer);
         // inc step counter
        _rStep := _rStep + 1;
       ELSE
         // check error ?
         IF (_writeLoadData.Error)
         THEN
           ErrorID     := _writeLoadData.ErrorID;
           ErrorAddTxt := _writeLoadData.ErrorAddTxt;;
         END_IF

         // timeout exceeded ?
         IF (CheckTimeout(_rTimer) = RobotLibraryConstants.OK)
         THEN
           ErrorID     := RobotLibraryErrorIdEnum.ERR_TIMEOUT_CMD;
           ErrorAddTxt := CONCAT(_stepName, DINT_TO_STRING(_rStep));
         END_IF
       END_IF

       // Wait Load data written ?
    5: IF (( NOT _writeLoadData.Busy  ) AND
           ( NOT _writeLoadData.Error ) AND
           (     _writeLoadData.Done  ))
       THEN
         // execute command
        _writeLoadData.Execute := FALSE;
         // apply Load data to internal Load data
        _loadData[_rSyncIdx] := LoadData[_rSyncIdx];
         // reset data changed bit
         AxesGroup.State.DataChanged.Load[_rSyncIdx] := FALSE;
         // dec count of unsynchronised Loads
         AxesGroup.State.SyncStatePlc.UnSyncNo.Load := AxesGroup.State.SyncStatePlc.UnSyncNo.Load - 1;
         // set timeout
         SetTimeout(PT := _rTimeout, rTimer := _rTimer);
         // dec step counter
        _rStep := _rStep - 2;
       ELSE
         // check error ?
         IF (_writeLoadData.Error)
         THEN
           WarningID := RobotLibraryWarningIdEnum.WARN_LOAD_SYNC_FAILED_BY_ERROR_OF_READ_OR_WRITE_CMD;
         END_IF

         // timeout exceeded ?
         IF (CheckTimeout(_rTimer) = RobotLibraryConstants.OK)
         THEN
           ErrorID     := RobotLibraryErrorIdEnum.ERR_TIMEOUT_CMD;
           ErrorAddTxt := CONCAT(_stepName, DINT_TO_STRING(_rStep));
         END_IF
       END_IF

    // --------------------------------------------
    // SyncMode after startup :
    // --------------------------------------------

    10 : // check synchronisation active ?
         IF ( AxesGroup.Parameter.Plc.Parameter.SynchronizationModes.Load[SyncTime.AFTER_START_UP] = SyncMode.NO_SYNCHRONIZATION)
         THEN
           RETURN;
         END_IF

         // reset count of unsynchronised Loads
         AxesGroup.State.SyncStatePlc.UnSyncNo.Load := 0;

         // Check all Load datas
         FOR _rSyncIdx := 1 TO AxesGroup.State.UnifiedLoadIndex //  !!! Attention : 0 is not allowed - LoadData starts with 1 !!!
         DO
           // compare Load data
           AxesGroup.State.DataChanged.Load[_rSyncIdx] := NOT IsLoadDataEqual( Data1 := LoadData[_rSyncIdx].Data, Data2 := _loadData[_rSyncIdx].Data, IgnoreTimestamp := FALSE);

           // Check Load data changed ?
           IF (AxesGroup.State.DataChanged.Load[_rSyncIdx])
           THEN
             // inc count of unsynchronised plc Loads
             AxesGroup.State.SyncStatePlc.UnSyncNo.Load := AxesGroup.State.SyncStatePlc.UnSyncNo.Load + 1;
             // Create log entry
             CreateLogMessagePara2 ( Timestamp   := SystemTime,
                                     MessageType := MessageType.CMD,
                                     Severity    := Severity.DEBUG,
                                     MessageCode := 0,
                                     MessageText := 'SyncLoadData: Detected a local change of Load[{1}] on PLC, SyncTime = {2}',
                                     Para1       :=  DINT_TO_STRING(_rSyncIdx),
                                     Para2       :=  SYNC_TIME_TO_STRING(SyncTime.AFTER_START_UP));
  				 END_IF

           // Update plc in sync flag
           AxesGroup.State.SyncStatePlc.InSync.Load := (AxesGroup.State.SyncStatePlc.UnSyncNo.Load = 0);
  	     END_FOR

         // Check synchronization is needed ?
         IF ( NOT AxesGroup.State.SyncStatePlc.InSync.Load ) XOR
            ( NOT AxesGroup.State.SyncStateRc .InSync.Load )
         THEN
           CASE AxesGroup.Parameter.Plc.Parameter.SynchronizationModes.Load[SyncTime.AFTER_START_UP]
           OF
             // NO_SYNCHRONIZATION
             SyncMode.NO_SYNCHRONIZATION : ; // no further action

             // CLIENT_TO_SERVER
             SyncMode.CLIENT_TO_SERVER :
               // set timeout
               SetTimeout(PT := _rTimeout, rTimer := _rTimer);
               // inc step counter
              _rStep := 11;

             // SERVER_TO_CLIENT
             SyncMode.SERVER_TO_CLIENT :
               // set timeout
               SetTimeout(PT := _rTimeout, rTimer := _rTimer);
               // inc step counter
              _rStep := 12;

             // AUTOMATIC
             SyncMode.AUTOMATIC :
               // set timeout
               SetTimeout(PT := _rTimeout, rTimer := _rTimer);
               // inc step counter
              _rStep := 13;
           END_CASE
         ELSE
           // datas changeḍ on both sides ? -> Warning
           IF (( NOT AxesGroup.State.SyncStatePlc.InSync.Load ) AND
               ( NOT AxesGroup.State.SyncStateRc .InSync.Load ))
           THEN
             WarningID := RobotLibraryWarningIdEnum.WARN_LOAD_SYNC_BOTH_SIDES_CHANGED;
           END_IF
         END_IF

    // ------------------------------------------
    // SyncMode : CLIENT_TO_SERVER
    // ------------------------------------------
    11 : // Conflict triggerd by PLC ?
         IF ( NOT AxesGroup.State.SyncStatePlc.InSync.Load )
         THEN
           // search for changed index
           FOR _rSyncIdx := 1 TO AxesGroup.State.UnifiedLoadIndex //  !!! Attention : 0 is not allowed - LoadData starts with 1 !!!
           DO
             IF ( AxesGroup.State.DataChanged.Load[_rSyncIdx] )
             THEN
               // set timeout
               SetTimeout(PT := _rTimeout, rTimer := _rTimer);
               // inc step counter
              _rStep := 30; // -> write PLC data to RC
               EXIT;
  					 END_IF
           END_FOR

           // Create log entry
           CreateLogMessagePara3 ( Timestamp   := SystemTime,
                                   MessageType := MessageType.CMD,
                                   Severity    := Severity.DEBUG,
                                   MessageCode := 0,
                                   MessageText := 'SyncLoadData: Synchronization of Load[{1}] triggered by PLC, SyncMode = {2}, SyncTime = {3}, SyncDirection = PLC -> RC',
                                   Para1       :=  DINT_TO_STRING(_rSyncIdx),
                                   Para2       :=  SYNC_MODE_TO_STRING(AxesGroup.Parameter.Plc.Parameter.SynchronizationModes.Load[SyncTime.AFTER_START_UP]),
                                   Para3       :=  SYNC_TIME_TO_STRING(SyncTime.AFTER_START_UP));
                                   RETURN;
         END_IF

         // Conflict triggered by RC ?
         IF ( NOT AxesGroup.State.SyncStateRc.InSync.Load )
         THEN
           // get changed index
          _rSyncIdx :=  LIMIT(1, AxesGroup.State.SyncStateRc.UnSyncNo.Load, AxesGroup.State.UnifiedLoadIndex); //  !!! Attention : 0 is not allowed - LoadData starts with 1 !!!
           // set timeout
           SetTimeout(PT := _rTimeout, rTimer := _rTimer);
           // inc step counter
          _rStep := 30; // -> write PLC data to RC

           // Create log entry
           CreateLogMessagePara3 ( Timestamp   := SystemTime,
                                   MessageType := MessageType.CMD,
                                   Severity    := Severity.DEBUG,
                                   MessageCode := 0,
                                   MessageText := 'SyncLoadData: Synchronization of Load[{1}] triggered by RC, SyncMode = {2}, SyncTime = {3}, SyncDirection = PLC -> RC',
                                   Para1       :=  DINT_TO_STRING(_rSyncIdx),
                                   Para2       :=  SYNC_MODE_TO_STRING(AxesGroup.Parameter.Plc.Parameter.SynchronizationModes.Load[SyncTime.AFTER_START_UP]),
                                   Para3       :=  SYNC_TIME_TO_STRING(SyncTime.AFTER_START_UP));
                                   RETURN;
  			 END_IF

         // set timeout
         SetTimeout(PT := _rTimeout, rTimer := _rTimer);
         // jump back
        _rStep := 10;

    // ------------------------------------------
    // SyncMode : SERVER_TO_CLIENT
    // ------------------------------------------
    12 : // Conflict triggerd by PLC ?
         IF ( NOT AxesGroup.State.SyncStatePlc.InSync.Load )
         THEN
           // search for changed index
           FOR _rSyncIdx := 1 TO AxesGroup.State.UnifiedLoadIndex //  !!! Attention : 0 is not allowed - LoadData starts with 1 !!!
           DO
             IF ( AxesGroup.State.DataChanged.Load[_rSyncIdx] )
             THEN
               // set timeout
               SetTimeout(PT := _rTimeout, rTimer := _rTimer);
               // inc step counter
              _rStep := 20; // -> read RC data and write it to PLC
               EXIT;
  					 END_IF
           END_FOR

           // Create log entry
           CreateLogMessagePara3 ( Timestamp   := SystemTime,
                                   MessageType := MessageType.CMD,
                                   Severity    := Severity.DEBUG,
                                   MessageCode := 0,
                                   MessageText := 'SyncLoadData: Synchronization of Load[{1}] triggered by PLC, SyncMode = {2}, SyncTime = {3}, SyncDirection = RC -> PLC',
                                   Para1       :=  DINT_TO_STRING(_rSyncIdx),
                                   Para2       :=  SYNC_MODE_TO_STRING(AxesGroup.Parameter.Plc.Parameter.SynchronizationModes.Load[SyncTime.AFTER_START_UP]),
                                   Para3       :=  SYNC_TIME_TO_STRING(SyncTime.AFTER_START_UP));
                                   RETURN;
         END_IF

         // Conflict triggered by RC ?
         IF ( NOT AxesGroup.State.SyncStateRc.InSync.Load )
         THEN
           // get changed index
          _rSyncIdx := LIMIT(1, AxesGroup.State.SyncStateRc.UnSyncNo.Load, AxesGroup.State.UnifiedLoadIndex); //  !!! Attention : 0 is not allowed - LoadData starts with 1 !!!
           // set timeout
           SetTimeout(PT := _rTimeout, rTimer := _rTimer);
           // inc step counter
          _rStep := 20; // -> read RC data and write it to PLC

           // Create log entry
           CreateLogMessagePara3 ( Timestamp   := SystemTime,
                                   MessageType := MessageType.CMD,
                                   Severity    := Severity.DEBUG,
                                   MessageCode := 0,
                                   MessageText := 'SyncLoadData: Synchronization of Load[{1}] triggered by RC, SyncMode = {2}, SyncTime = {3}, SyncDirection = RC -> PLC',
                                   Para1       :=  DINT_TO_STRING(_rSyncIdx),
                                   Para2       :=  SYNC_MODE_TO_STRING(AxesGroup.Parameter.Plc.Parameter.SynchronizationModes.Load[SyncTime.AFTER_START_UP]),
                                   Para3       :=  SYNC_TIME_TO_STRING(SyncTime.AFTER_START_UP));
                                   RETURN;
  			 END_IF

         // set timeout
         SetTimeout(PT := _rTimeout, rTimer := _rTimer);
         // jump back
        _rStep := 10;

    // ------------------------------------------
    // SyncMode : AUTOMATIC
    // ------------------------------------------
    13 : // Conflict triggerd by PLC ?
         IF ( NOT AxesGroup.State.SyncStatePlc.InSync.Load )
         THEN
           // search for changed index
           FOR _rSyncIdx := 1 TO AxesGroup.State.UnifiedLoadIndex //  !!! Attention : 0 is not allowed - LoadData starts with 1 !!!
           DO
             IF ( AxesGroup.State.DataChanged.Load[_rSyncIdx] )
             THEN
               // set timeout
               SetTimeout(PT := _rTimeout, rTimer := _rTimer);
               // inc step counter
              _rStep := 30; // -> write PLC data to RC
               EXIT;
  					 END_IF
           END_FOR
